//=============================================================================
// ST10_Flow15_FRobot_3.scl
// 1:1 CONVERSION FROM TIA PORTAL V18 GRAPH XML
// Generated: 2026-02-02
//=============================================================================

TYPE
    E_STEP_ST10_Flow15_FRobot_3 : (
        STEP_ST10_Flow15_FRobot_3_WaitRobotGripStatus := 360,
        STEP_ST10_Flow15_FRobot_3_WaitRobotFinish_4 := 356,
        STEP_ST10_Flow15_FRobot_3_ReqRobotToHomePos := 707,
        STEP_ST10_Flow15_FRobot_3_WaitRobotGripStatus_6 := 378,
        STEP_ST10_Flow15_FRobot_3_Tablecode_ScanFinish := 149,
        STEP_ST10_Flow15_FRobot_3_Open_NG_BOX_REQUESTED_ := 111,
        STEP_ST10_Flow15_FRobot_3_RobotReady_ := 311,
        STEP_ST10_Flow15_FRobot_3_PickPalletProcess := 250,
        STEP_ST10_Flow15_FRobot_3_WaitRobotFinish_9 := 371,
        STEP_ST10_Flow15_FRobot_3_WaitRobotReachPos4 := 318,
        STEP_ST10_Flow15_FRobot_3_WaitRobotStartHome := 383,
        STEP_ST10_Flow15_FRobot_3_RobotAutoCycle := 329,
        STEP_ST10_Flow15_FRobot_3_NG3_PutProcessFinish := 849,
        STEP_ST10_Flow15_FRobot_3_WaitRobotFinish_8 := 368,
        STEP_ST10_Flow15_FRobot_3_RobotScanGripperReachPos4 := 341,
        STEP_ST10_Flow15_FRobot_3_Step930 := 930,
        STEP_ST10_Flow15_FRobot_3_DataMove_6 := 266,
        STEP_ST10_Flow15_FRobot_3_ScanRing := 135,
        STEP_ST10_Flow15_FRobot_3_WaitRobotFinish_11 := 377,
        STEP_ST10_Flow15_FRobot_3_WaitRobotGripHaveStatus_2 := 348,
        STEP_ST10_Flow15_FRobot_3_WaitRobotGripStatus_3 := 369,
        STEP_ST10_Flow15_FRobot_3_S9 := 9,
        STEP_ST10_Flow15_FRobot_3_PartOKStatus := 249,
        STEP_ST10_Flow15_FRobot_3_WaitGripperPos3ScanFinish := 340,
        STEP_ST10_Flow15_FRobot_3_WaitBrakeTestFinish := 921,
        STEP_ST10_Flow15_FRobot_3_NG2_PutProcessFinish := 799,
        STEP_ST10_Flow15_FRobot_3_PressPick := 150,
        STEP_ST10_Flow15_FRobot_3_DataMove_2 := 257,
        STEP_ST10_Flow15_FRobot_3_DataMove_5 := 264,
        STEP_ST10_Flow15_FRobot_3_WaitRobotFinish := 327,
        STEP_ST10_Flow15_FRobot_3_StartRobotGluePut := 367,
        STEP_ST10_Flow15_FRobot_3_NG2Put_1Press_Glue := 160,
        STEP_ST10_Flow15_FRobot_3_F15_Initial := 1,
        STEP_ST10_Flow15_FRobot_3_BrakeTestFinish := 929,
        STEP_ST10_Flow15_FRobot_3_StartRobotNG2Put_1 := 373,
        STEP_ST10_Flow15_FRobot_3_NG2Put_2_Magnet := 165,
        STEP_ST10_Flow15_FRobot_3_WaitPos4ScanFinish := 319,
        STEP_ST10_Flow15_FRobot_3_PartOKStatus_1 := 273,
        STEP_ST10_Flow15_FRobot_3_WaitR1HomePosFinsh_1 := 899,
        STEP_ST10_Flow15_FRobot_3_RobotScanGripperReachPos2 := 337,
        STEP_ST10_Flow15_FRobot_3_StartRobotPickGlueNG := 328,
        STEP_ST10_Flow15_FRobot_3_PressRingPutProcessFinish := 599,
        STEP_ST10_Flow15_FRobot_3_StartRobotScanGripperCode := 334,
        STEP_ST10_Flow15_FRobot_3_DataMove_7 := 270,
        STEP_ST10_Flow15_FRobot_3_Maintenance := 131,
        STEP_ST10_Flow15_FRobot_3_Grip1PartStatus := 243,
        STEP_ST10_Flow15_FRobot_3_Grip1SensorError := 381,
        STEP_ST10_Flow15_FRobot_3_WaitMasteringTestFinish := 911,
        STEP_ST10_Flow15_FRobot_3_DataMove_4 := 262,
        STEP_ST10_Flow15_FRobot_3_PressShaftPut := 140,
        STEP_ST10_Flow15_FRobot_3_WaitRobotFinish_5 := 359,
        STEP_ST10_Flow15_FRobot_3_WaitRobotGripHaveStatus := 346,
        STEP_ST10_Flow15_FRobot_3_WaitRobotFinish_1 := 343,
        STEP_ST10_Flow15_FRobot_3_WaitGripperPos1ScanFinish := 336,
        STEP_ST10_Flow15_FRobot_3_RobotStart := 316,
        STEP_ST10_Flow15_FRobot_3_WaitPos2ScanFinish := 312,
        STEP_ST10_Flow15_FRobot_3_WaitRobotReachPos2 := 313,
        STEP_ST10_Flow15_FRobot_3_RobotHome := 317,
        STEP_ST10_Flow15_FRobot_3_WaitGripperPos4ScanFinish := 342,
        STEP_ST10_Flow15_FRobot_3_WaitScanCompletely := 247,
        STEP_ST10_Flow15_FRobot_3_PickGlueNGFinish_1 := 349,
        STEP_ST10_Flow15_FRobot_3_Grip2PartStatus := 244,
        STEP_ST10_Flow15_FRobot_3_WaitRobotFinish_3 := 353,
        STEP_ST10_Flow15_FRobot_3_WaitRobotGripStatus_1 := 363,
        STEP_ST10_Flow15_FRobot_3_NG2Put_3_Ring := 170,
        STEP_ST10_Flow15_FRobot_3_FlagReset := 272,
        STEP_ST10_Flow15_FRobot_3_WaitRobotGripStatus_2 := 366,
        STEP_ST10_Flow15_FRobot_3_WaitRobotFinish_6 := 362,
        STEP_ST10_Flow15_FRobot_3_Gripe2StatusAlarm := 332,
        STEP_ST10_Flow15_FRobot_3_DataMove_8 := 271,
        STEP_ST10_Flow15_FRobot_3_StartRobotPickTable := 352,
        STEP_ST10_Flow15_FRobot_3_ScanStart := 246,
        STEP_ST10_Flow15_FRobot_3_PickGlueNGReq := 120,
        STEP_ST10_Flow15_FRobot_3_RobotSpeed := 4,
        STEP_ST10_Flow15_FRobot_3_StartRobotPressPick := 364,
        STEP_ST10_Flow15_FRobot_3_MES_Online__offline_ := 385,
        STEP_ST10_Flow15_FRobot_3_S10_InitialFinish := 10,
        STEP_ST10_Flow15_FRobot_3_PickMagnScanNGBufferFinish := 399,
        STEP_ST10_Flow15_FRobot_3_RobotScanGripperReachPos3 := 339,
        STEP_ST10_Flow15_FRobot_3_GripStatusCheck := 330,
        STEP_ST10_Flow15_FRobot_3_ScanRingProcess := 450,
        STEP_ST10_Flow15_FRobot_3_S3 := 3,
        STEP_ST10_Flow15_FRobot_3_NG_2_PutProcess := 750,
        STEP_ST10_Flow15_FRobot_3_WaitRobotFinish_10 := 374,
        STEP_ST10_Flow15_FRobot_3_GluePutProcess := 650,
        STEP_ST10_Flow15_FRobot_3_PickTableProcessFinish := 449,
        STEP_ST10_Flow15_FRobot_3_DataClear := 252,
        STEP_ST10_Flow15_FRobot_3_Data_Clear_2 := 258,
        STEP_ST10_Flow15_FRobot_3_PickMagnetNGReqPick := 125,
        STEP_ST10_Flow15_FRobot_3_PressRingPutProcess := 550,
        STEP_ST10_Flow15_FRobot_3_WaitRobotFinish_2 := 345,
        STEP_ST10_Flow15_FRobot_3_PickTableProcess := 400,
        STEP_ST10_Flow15_FRobot_3_WaitRobotGripHaveStatus_3 := 354,
        STEP_ST10_Flow15_FRobot_3_NG_PutProcess := 700,
        STEP_ST10_Flow15_FRobot_3_StartRobotNGPut := 370,
        STEP_ST10_Flow15_FRobot_3_WaitRobotReachPos3 := 314,
        STEP_ST10_Flow15_FRobot_3_Maintenance_Pos := 850,
        STEP_ST10_Flow15_FRobot_3_PressPickProcess := 600,
        STEP_ST10_Flow15_FRobot_3_Data_Clear_9 := 269,
        STEP_ST10_Flow15_FRobot_3_PressPickProcessFinish_ := 649,
        STEP_ST10_Flow15_FRobot_3_WaitGripperPos2ScanFinish := 338,
        STEP_ST10_Flow15_FRobot_3_Tablecode_Scan := 200,
        STEP_ST10_Flow15_FRobot_3_MasteringTest_Req := 910,
        STEP_ST10_Flow15_FRobot_3_ProcessStart := 100,
        STEP_ST10_Flow15_FRobot_3_PartNGStatus := 251,
        STEP_ST10_Flow15_FRobot_3_Data_Clear_8 := 268,
        STEP_ST10_Flow15_FRobot_3_RobotManuallyMoved_ := 384,
        STEP_ST10_Flow15_FRobot_3_S5_MESInitial := 5,
        STEP_ST10_Flow15_FRobot_3_WaitRobotHomeRequest := 706,
        STEP_ST10_Flow15_FRobot_3_Masref_test := 132,
        STEP_ST10_Flow15_FRobot_3_BrakeTest_Req := 920,
        STEP_ST10_Flow15_FRobot_3_WaitRobotGripStatus_5 := 375,
        STEP_ST10_Flow15_FRobot_3_Data_Clear_4 := 261,
        STEP_ST10_Flow15_FRobot_3_ScanRingProcessFinish := 499,
        STEP_ST10_Flow15_FRobot_3_StartRobotPressShaftPut := 358,
        STEP_ST10_Flow15_FRobot_3_WaitPos1ScanFinish := 310,
        STEP_ST10_Flow15_FRobot_3_StartRobotScanFixtureCode := 308,
        STEP_ST10_Flow15_FRobot_3_StartRobotPickMagnScanNG := 344,
        STEP_ST10_Flow15_FRobot_3_ScanFixtureCode := 110,
        STEP_ST10_Flow15_FRobot_3_PressRingPut := 145,
        STEP_ST10_Flow15_FRobot_3_PickPallet := 115,
        STEP_ST10_Flow15_FRobot_3_WaitPos3ScanFinish := 315,
        STEP_ST10_Flow15_FRobot_3_WaitRobotReachScanPos := 357,
        STEP_ST10_Flow15_FRobot_3_StartRobotPressRingPut := 361,
        STEP_ST10_Flow15_FRobot_3_ReqRobotToMantenPos_1 := 704,
        STEP_ST10_Flow15_FRobot_3_PickTable := 130,
        STEP_ST10_Flow15_FRobot_3_DataMove_3 := 260,
        STEP_ST10_Flow15_FRobot_3_PickGlueNGProcess := 300,
        STEP_ST10_Flow15_FRobot_3_StartRobotPickPalletShaft := 326,
        STEP_ST10_Flow15_FRobot_3_NG1_PutProcessFinish := 749,
        STEP_ST10_Flow15_FRobot_3_OKPut := 155,
        STEP_ST10_Flow15_FRobot_3_PickPalletFinish := 299,
        STEP_ST10_Flow15_FRobot_3_MagnScanNGProcess := 350,
        STEP_ST10_Flow15_FRobot_3_OKPutProcessFinish := 699,
        STEP_ST10_Flow15_FRobot_3_StartRobotScanRing := 355,
        STEP_ST10_Flow15_FRobot_3_PressShaftPutProcessFinish := 549,
        STEP_ST10_Flow15_FRobot_3_DataMove_1 := 255,
        STEP_ST10_Flow15_FRobot_3_Grip2SensorError := 382,
        STEP_ST10_Flow15_FRobot_3_DataMove := 253,
        STEP_ST10_Flow15_FRobot_3_MasteringTestFinish := 919,
        STEP_ST10_Flow15_FRobot_3_S_900 := 900,
        STEP_ST10_Flow15_FRobot_3_WaitRobotReachPos1 := 309,
        STEP_ST10_Flow15_FRobot_3_RobotScanGripperReachPos1 := 335,
        STEP_ST10_Flow15_FRobot_3_Data_Clear_7 := 267,
        STEP_ST10_Flow15_FRobot_3_WaitR1MaintenPosFinsh_1 := 705,
        STEP_ST10_Flow15_FRobot_3_PressShaftPutProcess := 500,
        STEP_ST10_Flow15_FRobot_3_StartRobotNG3Put := 376,
        STEP_ST10_Flow15_FRobot_3_RobotTaskSelect := 333,
        STEP_ST10_Flow15_FRobot_3_NG_3_PutProcess := 800,
        STEP_ST10_Flow15_FRobot_3_Brake_Test := 133,
        STEP_ST10_Flow15_FRobot_3_WaitRobotFinish_7 := 365,
        STEP_ST10_Flow15_FRobot_3_Gripe1StatusAlarm := 331,
        STEP_ST10_Flow15_FRobot_3_WaitRobotGripStatus_4 := 372,
        STEP_ST10_Flow15_FRobot_3_Data_Clear_6 := 265,
        STEP_ST10_Flow15_FRobot_3_S2 := 2,
        STEP_ST10_Flow15_FRobot_3_CheckScanReady := 245,
        STEP_ST10_Flow15_FRobot_3_S8 := 8,
        STEP_ST10_Flow15_FRobot_3_CodeMove := 248,
        STEP_ST10_Flow15_FRobot_3_WaitRobotGripHaveStatus_1 := 347,
    ) INT := 1;
END_TYPE

CONST
    STEP_ST10_Flow15_FRobot_3_WaitRobotGripStatus := 360;
    STEP_ST10_Flow15_FRobot_3_WaitRobotFinish_4 := 356;
    STEP_ST10_Flow15_FRobot_3_ReqRobotToHomePos := 707;
    STEP_ST10_Flow15_FRobot_3_WaitRobotGripStatus_6 := 378;
    STEP_ST10_Flow15_FRobot_3_Tablecode_ScanFinish := 149;
    STEP_ST10_Flow15_FRobot_3_Open_NG_BOX_REQUESTED_ := 111;
    STEP_ST10_Flow15_FRobot_3_RobotReady_ := 311;
    STEP_ST10_Flow15_FRobot_3_PickPalletProcess := 250;
    STEP_ST10_Flow15_FRobot_3_WaitRobotFinish_9 := 371;
    STEP_ST10_Flow15_FRobot_3_WaitRobotReachPos4 := 318;
    STEP_ST10_Flow15_FRobot_3_WaitRobotStartHome := 383;
    STEP_ST10_Flow15_FRobot_3_RobotAutoCycle := 329;
    STEP_ST10_Flow15_FRobot_3_NG3_PutProcessFinish := 849;
    STEP_ST10_Flow15_FRobot_3_WaitRobotFinish_8 := 368;
    STEP_ST10_Flow15_FRobot_3_RobotScanGripperReachPos4 := 341;
    STEP_ST10_Flow15_FRobot_3_Step930 := 930;
    STEP_ST10_Flow15_FRobot_3_DataMove_6 := 266;
    STEP_ST10_Flow15_FRobot_3_ScanRing := 135;
    STEP_ST10_Flow15_FRobot_3_WaitRobotFinish_11 := 377;
    STEP_ST10_Flow15_FRobot_3_WaitRobotGripHaveStatus_2 := 348;
    STEP_ST10_Flow15_FRobot_3_WaitRobotGripStatus_3 := 369;
    STEP_ST10_Flow15_FRobot_3_S9 := 9;
    STEP_ST10_Flow15_FRobot_3_PartOKStatus := 249;
    STEP_ST10_Flow15_FRobot_3_WaitGripperPos3ScanFinish := 340;
    STEP_ST10_Flow15_FRobot_3_WaitBrakeTestFinish := 921;
    STEP_ST10_Flow15_FRobot_3_NG2_PutProcessFinish := 799;
    STEP_ST10_Flow15_FRobot_3_PressPick := 150;
    STEP_ST10_Flow15_FRobot_3_DataMove_2 := 257;
    STEP_ST10_Flow15_FRobot_3_DataMove_5 := 264;
    STEP_ST10_Flow15_FRobot_3_WaitRobotFinish := 327;
    STEP_ST10_Flow15_FRobot_3_StartRobotGluePut := 367;
    STEP_ST10_Flow15_FRobot_3_NG2Put_1Press_Glue := 160;
    STEP_ST10_Flow15_FRobot_3_F15_Initial := 1;
    STEP_ST10_Flow15_FRobot_3_BrakeTestFinish := 929;
    STEP_ST10_Flow15_FRobot_3_StartRobotNG2Put_1 := 373;
    STEP_ST10_Flow15_FRobot_3_NG2Put_2_Magnet := 165;
    STEP_ST10_Flow15_FRobot_3_WaitPos4ScanFinish := 319;
    STEP_ST10_Flow15_FRobot_3_PartOKStatus_1 := 273;
    STEP_ST10_Flow15_FRobot_3_WaitR1HomePosFinsh_1 := 899;
    STEP_ST10_Flow15_FRobot_3_RobotScanGripperReachPos2 := 337;
    STEP_ST10_Flow15_FRobot_3_StartRobotPickGlueNG := 328;
    STEP_ST10_Flow15_FRobot_3_PressRingPutProcessFinish := 599;
    STEP_ST10_Flow15_FRobot_3_StartRobotScanGripperCode := 334;
    STEP_ST10_Flow15_FRobot_3_DataMove_7 := 270;
    STEP_ST10_Flow15_FRobot_3_Maintenance := 131;
    STEP_ST10_Flow15_FRobot_3_Grip1PartStatus := 243;
    STEP_ST10_Flow15_FRobot_3_Grip1SensorError := 381;
    STEP_ST10_Flow15_FRobot_3_WaitMasteringTestFinish := 911;
    STEP_ST10_Flow15_FRobot_3_DataMove_4 := 262;
    STEP_ST10_Flow15_FRobot_3_PressShaftPut := 140;
    STEP_ST10_Flow15_FRobot_3_WaitRobotFinish_5 := 359;
    STEP_ST10_Flow15_FRobot_3_WaitRobotGripHaveStatus := 346;
    STEP_ST10_Flow15_FRobot_3_WaitRobotFinish_1 := 343;
    STEP_ST10_Flow15_FRobot_3_WaitGripperPos1ScanFinish := 336;
    STEP_ST10_Flow15_FRobot_3_RobotStart := 316;
    STEP_ST10_Flow15_FRobot_3_WaitPos2ScanFinish := 312;
    STEP_ST10_Flow15_FRobot_3_WaitRobotReachPos2 := 313;
    STEP_ST10_Flow15_FRobot_3_RobotHome := 317;
    STEP_ST10_Flow15_FRobot_3_WaitGripperPos4ScanFinish := 342;
    STEP_ST10_Flow15_FRobot_3_WaitScanCompletely := 247;
    STEP_ST10_Flow15_FRobot_3_PickGlueNGFinish_1 := 349;
    STEP_ST10_Flow15_FRobot_3_Grip2PartStatus := 244;
    STEP_ST10_Flow15_FRobot_3_WaitRobotFinish_3 := 353;
    STEP_ST10_Flow15_FRobot_3_WaitRobotGripStatus_1 := 363;
    STEP_ST10_Flow15_FRobot_3_NG2Put_3_Ring := 170;
    STEP_ST10_Flow15_FRobot_3_FlagReset := 272;
    STEP_ST10_Flow15_FRobot_3_WaitRobotGripStatus_2 := 366;
    STEP_ST10_Flow15_FRobot_3_WaitRobotFinish_6 := 362;
    STEP_ST10_Flow15_FRobot_3_Gripe2StatusAlarm := 332;
    STEP_ST10_Flow15_FRobot_3_DataMove_8 := 271;
    STEP_ST10_Flow15_FRobot_3_StartRobotPickTable := 352;
    STEP_ST10_Flow15_FRobot_3_ScanStart := 246;
    STEP_ST10_Flow15_FRobot_3_PickGlueNGReq := 120;
    STEP_ST10_Flow15_FRobot_3_RobotSpeed := 4;
    STEP_ST10_Flow15_FRobot_3_StartRobotPressPick := 364;
    STEP_ST10_Flow15_FRobot_3_MES_Online__offline_ := 385;
    STEP_ST10_Flow15_FRobot_3_S10_InitialFinish := 10;
    STEP_ST10_Flow15_FRobot_3_PickMagnScanNGBufferFinish := 399;
    STEP_ST10_Flow15_FRobot_3_RobotScanGripperReachPos3 := 339;
    STEP_ST10_Flow15_FRobot_3_GripStatusCheck := 330;
    STEP_ST10_Flow15_FRobot_3_ScanRingProcess := 450;
    STEP_ST10_Flow15_FRobot_3_S3 := 3;
    STEP_ST10_Flow15_FRobot_3_NG_2_PutProcess := 750;
    STEP_ST10_Flow15_FRobot_3_WaitRobotFinish_10 := 374;
    STEP_ST10_Flow15_FRobot_3_GluePutProcess := 650;
    STEP_ST10_Flow15_FRobot_3_PickTableProcessFinish := 449;
    STEP_ST10_Flow15_FRobot_3_DataClear := 252;
    STEP_ST10_Flow15_FRobot_3_Data_Clear_2 := 258;
    STEP_ST10_Flow15_FRobot_3_PickMagnetNGReqPick := 125;
    STEP_ST10_Flow15_FRobot_3_PressRingPutProcess := 550;
    STEP_ST10_Flow15_FRobot_3_WaitRobotFinish_2 := 345;
    STEP_ST10_Flow15_FRobot_3_PickTableProcess := 400;
    STEP_ST10_Flow15_FRobot_3_WaitRobotGripHaveStatus_3 := 354;
    STEP_ST10_Flow15_FRobot_3_NG_PutProcess := 700;
    STEP_ST10_Flow15_FRobot_3_StartRobotNGPut := 370;
    STEP_ST10_Flow15_FRobot_3_WaitRobotReachPos3 := 314;
    STEP_ST10_Flow15_FRobot_3_Maintenance_Pos := 850;
    STEP_ST10_Flow15_FRobot_3_PressPickProcess := 600;
    STEP_ST10_Flow15_FRobot_3_Data_Clear_9 := 269;
    STEP_ST10_Flow15_FRobot_3_PressPickProcessFinish_ := 649;
    STEP_ST10_Flow15_FRobot_3_WaitGripperPos2ScanFinish := 338;
    STEP_ST10_Flow15_FRobot_3_Tablecode_Scan := 200;
    STEP_ST10_Flow15_FRobot_3_MasteringTest_Req := 910;
    STEP_ST10_Flow15_FRobot_3_ProcessStart := 100;
    STEP_ST10_Flow15_FRobot_3_PartNGStatus := 251;
    STEP_ST10_Flow15_FRobot_3_Data_Clear_8 := 268;
    STEP_ST10_Flow15_FRobot_3_RobotManuallyMoved_ := 384;
    STEP_ST10_Flow15_FRobot_3_S5_MESInitial := 5;
    STEP_ST10_Flow15_FRobot_3_WaitRobotHomeRequest := 706;
    STEP_ST10_Flow15_FRobot_3_Masref_test := 132;
    STEP_ST10_Flow15_FRobot_3_BrakeTest_Req := 920;
    STEP_ST10_Flow15_FRobot_3_WaitRobotGripStatus_5 := 375;
    STEP_ST10_Flow15_FRobot_3_Data_Clear_4 := 261;
    STEP_ST10_Flow15_FRobot_3_ScanRingProcessFinish := 499;
    STEP_ST10_Flow15_FRobot_3_StartRobotPressShaftPut := 358;
    STEP_ST10_Flow15_FRobot_3_WaitPos1ScanFinish := 310;
    STEP_ST10_Flow15_FRobot_3_StartRobotScanFixtureCode := 308;
    STEP_ST10_Flow15_FRobot_3_StartRobotPickMagnScanNG := 344;
    STEP_ST10_Flow15_FRobot_3_ScanFixtureCode := 110;
    STEP_ST10_Flow15_FRobot_3_PressRingPut := 145;
    STEP_ST10_Flow15_FRobot_3_PickPallet := 115;
    STEP_ST10_Flow15_FRobot_3_WaitPos3ScanFinish := 315;
    STEP_ST10_Flow15_FRobot_3_WaitRobotReachScanPos := 357;
    STEP_ST10_Flow15_FRobot_3_StartRobotPressRingPut := 361;
    STEP_ST10_Flow15_FRobot_3_ReqRobotToMantenPos_1 := 704;
    STEP_ST10_Flow15_FRobot_3_PickTable := 130;
    STEP_ST10_Flow15_FRobot_3_DataMove_3 := 260;
    STEP_ST10_Flow15_FRobot_3_PickGlueNGProcess := 300;
    STEP_ST10_Flow15_FRobot_3_StartRobotPickPalletShaft := 326;
    STEP_ST10_Flow15_FRobot_3_NG1_PutProcessFinish := 749;
    STEP_ST10_Flow15_FRobot_3_OKPut := 155;
    STEP_ST10_Flow15_FRobot_3_PickPalletFinish := 299;
    STEP_ST10_Flow15_FRobot_3_MagnScanNGProcess := 350;
    STEP_ST10_Flow15_FRobot_3_OKPutProcessFinish := 699;
    STEP_ST10_Flow15_FRobot_3_StartRobotScanRing := 355;
    STEP_ST10_Flow15_FRobot_3_PressShaftPutProcessFinish := 549;
    STEP_ST10_Flow15_FRobot_3_DataMove_1 := 255;
    STEP_ST10_Flow15_FRobot_3_Grip2SensorError := 382;
    STEP_ST10_Flow15_FRobot_3_DataMove := 253;
    STEP_ST10_Flow15_FRobot_3_MasteringTestFinish := 919;
    STEP_ST10_Flow15_FRobot_3_S_900 := 900;
    STEP_ST10_Flow15_FRobot_3_WaitRobotReachPos1 := 309;
    STEP_ST10_Flow15_FRobot_3_RobotScanGripperReachPos1 := 335;
    STEP_ST10_Flow15_FRobot_3_Data_Clear_7 := 267;
    STEP_ST10_Flow15_FRobot_3_WaitR1MaintenPosFinsh_1 := 705;
    STEP_ST10_Flow15_FRobot_3_PressShaftPutProcess := 500;
    STEP_ST10_Flow15_FRobot_3_StartRobotNG3Put := 376;
    STEP_ST10_Flow15_FRobot_3_RobotTaskSelect := 333;
    STEP_ST10_Flow15_FRobot_3_NG_3_PutProcess := 800;
    STEP_ST10_Flow15_FRobot_3_Brake_Test := 133;
    STEP_ST10_Flow15_FRobot_3_WaitRobotFinish_7 := 365;
    STEP_ST10_Flow15_FRobot_3_Gripe1StatusAlarm := 331;
    STEP_ST10_Flow15_FRobot_3_WaitRobotGripStatus_4 := 372;
    STEP_ST10_Flow15_FRobot_3_Data_Clear_6 := 265;
    STEP_ST10_Flow15_FRobot_3_S2 := 2;
    STEP_ST10_Flow15_FRobot_3_CheckScanReady := 245;
    STEP_ST10_Flow15_FRobot_3_S8 := 8;
    STEP_ST10_Flow15_FRobot_3_CodeMove := 248;
    STEP_ST10_Flow15_FRobot_3_WaitRobotGripHaveStatus_1 := 347;
END_CONST

FUNCTION_BLOCK "ST10_Flow15_FRobot_3_1to1"
{ S7_Optimized_Access := 'TRUE' }
VERSION : 1.0

VAR_INPUT
    iSysInface : "RCS_SysComInterface_V1";
END_VAR

VAR_IN_OUT
    ioPM_Inface : "RCS_PMInterface_V1";
    ioStatus : Int;
END_VAR

VAR_OUTPUT
    oAlarmID : Int;
END_VAR

VAR
    State : INT := 1;
    act_InitialRun : Bool;
    act_InitialOK : Bool;
    act_WaitRunning : Bool;
    act_Running : Bool;
    act_ProcessComplete : Bool;
    act_ProcessStart : Bool;
    act_UnPause : Bool;
    bError : Bool;
    wErrorID : Word;
END_VAR

BEGIN
    //======================================================================
    // STATE MACHINE - Inline Transition Conditions
    //======================================================================

    CASE #State OF

        // ===========================================
        // STEP 360: WaitRobotGripStatus
        // ===========================================
        STEP_ST10_Flow15_FRobot_3_WaitRobotGripStatus:
            // No actions in XML

            // Transition to next step: 356
            IF TRUE THEN  // Sequential transition - review XML for actual condition
                #State := STEP_ST10_Flow15_FRobot_3_WaitRobotFinish_4;
            END_IF;

        // ===========================================
        // STEP 356: WaitRobotFinish_4
        // ===========================================
        STEP_ST10_Flow15_FRobot_3_WaitRobotFinish_4:
            // Action Qualifier=N
            // Token: "KukaRobot3_CtrlDB".sPLCtoROB.User.Cycle.DI262_ScanRingComplete
            "KukaRobot3_CtrlDB".sPLCtoROB.User.Cycle.DI262_ScanRingComplete;

            // Transition to next step: 707
            IF TRUE THEN  // Sequential transition - review XML for actual condition
                #State := STEP_ST10_Flow15_FRobot_3_ReqRobotToHomePos;
            END_IF;

        // ===========================================
        // STEP 707: ReqRobotToHomePos
        // ===========================================
        STEP_ST10_Flow15_FRobot_3_ReqRobotToHomePos:
            // Action Qualifier=N
            // Token: "KukaRobot3_CtrlDB".sPLCtoROB.User.Cycle.DI300_HomeRequest
            "KukaRobot3_CtrlDB".sPLCtoROB.User.Cycle.DI300_HomeRequest;

            // Transition to next step: 378
            IF TRUE THEN  // Sequential transition - review XML for actual condition
                #State := STEP_ST10_Flow15_FRobot_3_WaitRobotGripStatus_6;
            END_IF;

        // ===========================================
        // STEP 378: WaitRobotGripStatus_6
        // ===========================================
        STEP_ST10_Flow15_FRobot_3_WaitRobotGripStatus_6:
            // No actions in XML

            // Transition to next step: 149
            IF TRUE THEN  // Sequential transition - review XML for actual condition
                #State := STEP_ST10_Flow15_FRobot_3_Tablecode_ScanFinish;
            END_IF;

        // ===========================================
        // STEP 149: Tablecode ScanFinish
        // ===========================================
        STEP_ST10_Flow15_FRobot_3_Tablecode_ScanFinish:
            // Action Qualifier=S
            // Token: #ioPM_Inface.ProcessComplete
            #ioPM_Inface.ProcessComplete := TRUE;
            // Action Qualifier=R
            // Token: #ioPM_Inface.ProcessStart
            #ioPM_Inface.ProcessStart := FALSE;

            // Transition to next step: 111
            IF TRUE THEN  // Sequential transition - review XML for actual condition
                #State := STEP_ST10_Flow15_FRobot_3_Open_NG_BOX_REQUESTED_;
            END_IF;

        // ===========================================
        // STEP 111: Open NG BOX REQUESTED?
        // ===========================================
        STEP_ST10_Flow15_FRobot_3_Open_NG_BOX_REQUESTED_:
            // No actions in XML

            // Transition to next step: 311
            IF TRUE THEN  // Sequential transition - review XML for actual condition
                #State := STEP_ST10_Flow15_FRobot_3_RobotReady_;
            END_IF;

        // ===========================================
        // STEP 311: RobotReady?
        // ===========================================
        STEP_ST10_Flow15_FRobot_3_RobotReady_:
            // No actions in XML

            // Transition to next step: 250
            IF TRUE THEN  // Sequential transition - review XML for actual condition
                #State := STEP_ST10_Flow15_FRobot_3_PickPalletProcess;
            END_IF;

        // ===========================================
        // STEP 250: PickPalletProcess
        // ===========================================
        STEP_ST10_Flow15_FRobot_3_PickPalletProcess:
            // No actions in XML

            // Transition to next step: 371
            IF TRUE THEN  // Sequential transition - review XML for actual condition
                #State := STEP_ST10_Flow15_FRobot_3_WaitRobotFinish_9;
            END_IF;

        // ===========================================
        // STEP 371: WaitRobotFinish_9
        // ===========================================
        STEP_ST10_Flow15_FRobot_3_WaitRobotFinish_9:
            // No actions in XML

            // Transition to next step: 318
            IF TRUE THEN  // Sequential transition - review XML for actual condition
                #State := STEP_ST10_Flow15_FRobot_3_WaitRobotReachPos4;
            END_IF;

        // ===========================================
        // STEP 318: WaitRobotReachPos4
        // ===========================================
        STEP_ST10_Flow15_FRobot_3_WaitRobotReachPos4:
            // No actions in XML

            // Transition to next step: 383
            IF TRUE THEN  // Sequential transition - review XML for actual condition
                #State := STEP_ST10_Flow15_FRobot_3_WaitRobotStartHome;
            END_IF;

        // ===========================================
        // STEP 383: WaitRobotStartHome
        // ===========================================
        STEP_ST10_Flow15_FRobot_3_WaitRobotStartHome:
            // No actions in XML

            // Transition to next step: 329
            IF TRUE THEN  // Sequential transition - review XML for actual condition
                #State := STEP_ST10_Flow15_FRobot_3_RobotAutoCycle;
            END_IF;

        // ===========================================
        // STEP 329: RobotAutoCycle
        // ===========================================
        STEP_ST10_Flow15_FRobot_3_RobotAutoCycle:
            // Action Qualifier=N
            // Token: "KukaRobot3_CtrlDB".ioStartAutoCycle
            "KukaRobot3_CtrlDB".ioStartAutoCycle;

            // Transition to next step: 849
            IF TRUE THEN  // Sequential transition - review XML for actual condition
                #State := STEP_ST10_Flow15_FRobot_3_NG3_PutProcessFinish;
            END_IF;

        // ===========================================
        // STEP 849: NG3 PutProcessFinish
        // ===========================================
        STEP_ST10_Flow15_FRobot_3_NG3_PutProcessFinish:
            // Action Qualifier=S
            // Token: #ioPM_Inface.ProcessComplete
            #ioPM_Inface.ProcessComplete := TRUE;
            // Action Qualifier=R
            // Token: #ioPM_Inface.ProcessStart
            #ioPM_Inface.ProcessStart := FALSE;

            // Transition to next step: 368
            IF TRUE THEN  // Sequential transition - review XML for actual condition
                #State := STEP_ST10_Flow15_FRobot_3_WaitRobotFinish_8;
            END_IF;

        // ===========================================
        // STEP 368: WaitRobotFinish_8
        // ===========================================
        STEP_ST10_Flow15_FRobot_3_WaitRobotFinish_8:
            // No actions in XML

            // Transition to next step: 341
            IF TRUE THEN  // Sequential transition - review XML for actual condition
                #State := STEP_ST10_Flow15_FRobot_3_RobotScanGripperReachPos4;
            END_IF;

        // ===========================================
        // STEP 341: RobotScanGripperReachPos4
        // ===========================================
        STEP_ST10_Flow15_FRobot_3_RobotScanGripperReachPos4:
            // No actions in XML

            // Transition to next step: 930
            IF TRUE THEN  // Sequential transition - review XML for actual condition
                #State := STEP_ST10_Flow15_FRobot_3_Step930;
            END_IF;

        // ===========================================
        // STEP 930: Step930
        // ===========================================
        STEP_ST10_Flow15_FRobot_3_Step930:
            // Action Qualifier=N
            // Token: //"AutoProcessData".F_Robot3Grip1.PartStatus:=444
            //"AutoProcessData".F_Robot3Grip1.PartStatus:=444;

            // Transition to next step: 266
            IF TRUE THEN  // Sequential transition - review XML for actual condition
                #State := STEP_ST10_Flow15_FRobot_3_DataMove_6;
            END_IF;

        // ===========================================
        // STEP 266: DataMove_6
        // ===========================================
        STEP_ST10_Flow15_FRobot_3_DataMove_6:
            // Action Qualifier=N
            // Token: //"AutoProcessData_Buffer".DataBuffer["AutoProcessData".GlobalData.DataIndex]:="AutoProcessData".F_Robot3Grip1
            //"AutoProcessData_Buffer".DataBuffer["AutoProcessData".GlobalData.DataIndex]:="AutoProcessData".F_Robot3Grip1;
            // Action Qualifier=N
            // Token: //"AutoProcessData".GlobalData.DataIndex:="AutoProcessData".GlobalData.DataIndex+1
            //"AutoProcessData".GlobalData.DataIndex:="AutoProcessData".GlobalData.DataIndex+1;

            // Transition to next step: 135
            IF TRUE THEN  // Sequential transition - review XML for actual condition
                #State := STEP_ST10_Flow15_FRobot_3_ScanRing;
            END_IF;

        // ===========================================
        // STEP 135: ScanRing
        // ===========================================
        STEP_ST10_Flow15_FRobot_3_ScanRing:
            // Action Qualifier=R
            // Token: #ioPM_Inface.ProcessComplete
            #ioPM_Inface.ProcessComplete := FALSE;
            // Action Qualifier=S
            // Token: #ioPM_Inface.ProcessStart
            #ioPM_Inface.ProcessStart := TRUE;

            // Transition to next step: 377
            IF TRUE THEN  // Sequential transition - review XML for actual condition
                #State := STEP_ST10_Flow15_FRobot_3_WaitRobotFinish_11;
            END_IF;

        // ===========================================
        // STEP 377: WaitRobotFinish_11
        // ===========================================
        STEP_ST10_Flow15_FRobot_3_WaitRobotFinish_11:
            // No actions in XML

            // Transition to next step: 348
            IF TRUE THEN  // Sequential transition - review XML for actual condition
                #State := STEP_ST10_Flow15_FRobot_3_WaitRobotGripHaveStatus_2;
            END_IF;

        // ===========================================
        // STEP 348: WaitRobotGripHaveStatus_2
        // ===========================================
        STEP_ST10_Flow15_FRobot_3_WaitRobotGripHaveStatus_2:
            // No actions in XML

            // Transition to next step: 369
            IF TRUE THEN  // Sequential transition - review XML for actual condition
                #State := STEP_ST10_Flow15_FRobot_3_WaitRobotGripStatus_3;
            END_IF;

        // ===========================================
        // STEP 369: WaitRobotGripStatus_3
        // ===========================================
        STEP_ST10_Flow15_FRobot_3_WaitRobotGripStatus_3:
            // No actions in XML

            // Transition to next step: 9
            IF TRUE THEN  // Sequential transition - review XML for actual condition
                #State := STEP_ST10_Flow15_FRobot_3_S9;
            END_IF;

        // ===========================================
        // STEP 9: S9
        // ===========================================
        STEP_ST10_Flow15_FRobot_3_S9:
            // No actions in XML

            // Transition to next step: 249
            IF TRUE THEN  // Sequential transition - review XML for actual condition
                #State := STEP_ST10_Flow15_FRobot_3_PartOKStatus;
            END_IF;

        // ===========================================
        // STEP 249: PartOKStatus
        // ===========================================
        STEP_ST10_Flow15_FRobot_3_PartOKStatus:
            // Action Qualifier=N
            // Token: "AutoProcessData".F_Robot3Grip2.PartStatus := 199
            "AutoProcessData".F_Robot3Grip2.PartStatus := 199;

            // Transition to next step: 340
            IF TRUE THEN  // Sequential transition - review XML for actual condition
                #State := STEP_ST10_Flow15_FRobot_3_WaitGripperPos3ScanFinish;
            END_IF;

        // ===========================================
        // STEP 340: WaitGripperPos3ScanFinish
        // ===========================================
        STEP_ST10_Flow15_FRobot_3_WaitGripperPos3ScanFinish:
            // No actions in XML

            // Transition to next step: 921
            IF TRUE THEN  // Sequential transition - review XML for actual condition
                #State := STEP_ST10_Flow15_FRobot_3_WaitBrakeTestFinish;
            END_IF;

        // ===========================================
        // STEP 921: WaitBrakeTestFinish
        // ===========================================
        STEP_ST10_Flow15_FRobot_3_WaitBrakeTestFinish:
            // No actions in XML

            // Transition to next step: 799
            IF TRUE THEN  // Sequential transition - review XML for actual condition
                #State := STEP_ST10_Flow15_FRobot_3_NG2_PutProcessFinish;
            END_IF;

        // ===========================================
        // STEP 799: NG2 PutProcessFinish
        // ===========================================
        STEP_ST10_Flow15_FRobot_3_NG2_PutProcessFinish:
            // Action Qualifier=S
            // Token: #ioPM_Inface.ProcessComplete
            #ioPM_Inface.ProcessComplete := TRUE;
            // Action Qualifier=R
            // Token: #ioPM_Inface.ProcessStart
            #ioPM_Inface.ProcessStart := FALSE;
            // Action Qualifier=N
            // Token: "AutoProcessData".F_Robot3Grip1.PartStatus := 0
            "AutoProcessData".F_Robot3Grip1.PartStatus := 0;

            // Transition to next step: 150
            IF TRUE THEN  // Sequential transition - review XML for actual condition
                #State := STEP_ST10_Flow15_FRobot_3_PressPick;
            END_IF;

        // ===========================================
        // STEP 150: PressPick
        // ===========================================
        STEP_ST10_Flow15_FRobot_3_PressPick:
            // Action Qualifier=R
            // Token: #ioPM_Inface.ProcessComplete
            #ioPM_Inface.ProcessComplete := FALSE;
            // Action Qualifier=S
            // Token: #ioPM_Inface.ProcessStart
            #ioPM_Inface.ProcessStart := TRUE;

            // Transition to next step: 257
            IF TRUE THEN  // Sequential transition - review XML for actual condition
                #State := STEP_ST10_Flow15_FRobot_3_DataMove_2;
            END_IF;

        // ===========================================
        // STEP 257: DataMove_2
        // ===========================================
        STEP_ST10_Flow15_FRobot_3_DataMove_2:
            // Action Qualifier=N, Event="S1"
            // Token: "AutoProcessData".B_Press2 := "AutoProcessData".F_Robot3Grip1
            "AutoProcessData".B_Press2 := "AutoProcessData".F_Robot3Grip1;
            // Action Qualifier=N, Event="S1"
            // Token: "AutoProcessData".F_Robot3Grip1 := "AutoProcessData".ClearData
            "AutoProcessData".F_Robot3Grip1 := "AutoProcessData".ClearData;

            // Transition to next step: 264
            IF TRUE THEN  // Sequential transition - review XML for actual condition
                #State := STEP_ST10_Flow15_FRobot_3_DataMove_5;
            END_IF;

        // ===========================================
        // STEP 264: DataMove_5
        // ===========================================
        STEP_ST10_Flow15_FRobot_3_DataMove_5:
            // Action Qualifier=N, Event="S1"
            // Token: "AutoProcessData_Buffer".DataBuffer["AutoProcessData".GlobalData.DataIndex] := "AutoProcessData".F_Robot3Grip1
            "AutoProcessData_Buffer".DataBuffer["AutoProcessData".GlobalData.DataIndex] := "AutoProcessData".F_Robot3Grip1;
            // Action Qualifier=N, Event="S1"
            // Token: "AutoProcessData".F_Robot3Grip1 := "AutoProcessData".ClearData
            "AutoProcessData".F_Robot3Grip1 := "AutoProcessData".ClearData;
            // Action Qualifier=N, Event="S0"
            // Token: "AutoProcessData".GlobalData.DataIndex := "AutoProcessData".GlobalData.DataIndex + 1
            "AutoProcessData".GlobalData.DataIndex := "AutoProcessData".GlobalData.DataIndex + 1;

            // Transition to next step: 327
            IF TRUE THEN  // Sequential transition - review XML for actual condition
                #State := STEP_ST10_Flow15_FRobot_3_WaitRobotFinish;
            END_IF;

        // ===========================================
        // STEP 327: WaitRobotFinish
        // ===========================================
        STEP_ST10_Flow15_FRobot_3_WaitRobotFinish:
            // No actions in XML

            // Transition to next step: 367
            IF TRUE THEN  // Sequential transition - review XML for actual condition
                #State := STEP_ST10_Flow15_FRobot_3_StartRobotGluePut;
            END_IF;

        // ===========================================
        // STEP 367: StartRobotGluePut
        // ===========================================
        STEP_ST10_Flow15_FRobot_3_StartRobotGluePut:
            // Action Qualifier=N
            // Token: "KukaRobot3_CtrlDB".sPLCtoROB.User.Cycle.DI289_PutOkPartReq
            "KukaRobot3_CtrlDB".sPLCtoROB.User.Cycle.DI289_PutOkPartReq;

            // Transition to next step: 160
            IF TRUE THEN  // Sequential transition - review XML for actual condition
                #State := STEP_ST10_Flow15_FRobot_3_NG2Put_1Press_Glue;
            END_IF;

        // ===========================================
        // STEP 160: NG2Put_1Press/Glue
        // ===========================================
        STEP_ST10_Flow15_FRobot_3_NG2Put_1Press_Glue:
            // Action Qualifier=R
            // Token: #ioPM_Inface.ProcessComplete
            #ioPM_Inface.ProcessComplete := FALSE;
            // Action Qualifier=S
            // Token: #ioPM_Inface.ProcessStart
            #ioPM_Inface.ProcessStart := TRUE;

            // Transition to next step: 1
            IF TRUE THEN  // Sequential transition - review XML for actual condition
                #State := STEP_ST10_Flow15_FRobot_3_F15_Initial;
            END_IF;

        // ===========================================
        // STEP 1: F15_Initial
        // ===========================================
        STEP_ST10_Flow15_FRobot_3_F15_Initial:
            // Action Qualifier=S
            // Token: #ioPM_Inface.InitialRun
            #ioPM_Inface.InitialRun := TRUE;
            // Action Qualifier=R
            // Token: #ioPM_Inface.InitialOK
            #ioPM_Inface.InitialOK := FALSE;
            // Action Qualifier=R
            // Token: #ioPM_Inface.WaitRunning
            #ioPM_Inface.WaitRunning := FALSE;
            // Action Qualifier=R
            // Token: #ioPM_Inface.Running
            #ioPM_Inface.Running := FALSE;
            // Action Qualifier=R
            // Token: #ioPM_Inface.ProcessComplete
            #ioPM_Inface.ProcessComplete := FALSE;
            // Action Qualifier=R
            // Token: #ioPM_Inface.UnPause
            #ioPM_Inface.UnPause := FALSE;
            // Action Qualifier=R
            // Token: "Station_Sys".Cmd.Calibration
            "Station_Sys".Cmd.Calibration := FALSE;
            // Action Qualifier=R
            // Token: "Station_Sys".Cmd.ChangeOver
            "Station_Sys".Cmd.ChangeOver := FALSE;
            // Action Qualifier=N
            // Token: //"ST350_Sys".Cmd.DryRun
            //"ST350_Sys".Cmd.DryRun;
            // Action Qualifier=R
            // Token: "Station_Sys".Cmd.Reserve
            "Station_Sys".Cmd.Reserve := FALSE;
            // Action Qualifier=R
            // Token: "Station_Sys".Cmd.OneCycle
            "Station_Sys".Cmd.OneCycle := FALSE;
            // Action Qualifier=R
            // Token: "AutoProcessControl".Robot_3.Press2PutFlag
            "AutoProcessControl".Robot_3.Press2PutFlag := FALSE;
            // Action Qualifier=R
            // Token: "AutoProcessControl".Robot_3.Press2PickFlag
            "AutoProcessControl".Robot_3.Press2PickFlag := FALSE;
            // Action Qualifier=R
            // Token: "AutoProcessControl".Robot_3.GlueNGPickFlag
            "AutoProcessControl".Robot_3.GlueNGPickFlag := FALSE;
            // Action Qualifier=R
            // Token: "AutoProcessControl".Robot_3.ScanNGPickFlag
            "AutoProcessControl".Robot_3.ScanNGPickFlag := FALSE;
            // Action Qualifier=R
            // Token: "AutoProcessControl".Robot_3.NGPutFlag
            "AutoProcessControl".Robot_3.NGPutFlag := FALSE;
            // Action Qualifier=R
            // Token: #ioPM_Inface.ProcessStart
            #ioPM_Inface.ProcessStart := FALSE;
            // Action Qualifier=R
            // Token: "ChangeOver_DB".Robot_3.MaintenancePosReqSelFlag
            "ChangeOver_DB".Robot_3.MaintenancePosReqSelFlag := FALSE;
            // Action Qualifier=N
            // Token: //"Robot_DB".Robot_3.MasteringTest_Req
            //"Robot_DB".Robot_3.MasteringTest_Req;
            // Action Qualifier=N
            // Token: //"Robot_DB".Robot_3.BrakeTest_Req
            //"Robot_DB".Robot_3.BrakeTest_Req;
            // Action Qualifier=R
            // Token: #Auto_Run_after_NG_box_closed
            #Auto_Run_after_NG_box_closed := FALSE;

            // Transition to next step: 929
            IF TRUE THEN  // Sequential transition - review XML for actual condition
                #State := STEP_ST10_Flow15_FRobot_3_BrakeTestFinish;
            END_IF;

        // ===========================================
        // STEP 929: BrakeTestFinish
        // ===========================================
        STEP_ST10_Flow15_FRobot_3_BrakeTestFinish:
            // Action Qualifier=R
            // Token: "Robot_DB".Robot_3.BrakeTest_Req
            "Robot_DB".Robot_3.BrakeTest_Req := FALSE;

            // Transition to next step: 373
            IF TRUE THEN  // Sequential transition - review XML for actual condition
                #State := STEP_ST10_Flow15_FRobot_3_StartRobotNG2Put_1;
            END_IF;

        // ===========================================
        // STEP 373: StartRobotNG2Put_1
        // ===========================================
        STEP_ST10_Flow15_FRobot_3_StartRobotNG2Put_1:
            // Action Qualifier=N
            // Token: "KukaRobot3_CtrlDB".sPLCtoROB.User.Cycle.DI266_LoadGlueNGReq2
            "KukaRobot3_CtrlDB".sPLCtoROB.User.Cycle.DI266_LoadGlueNGReq2;

            // Transition to next step: 165
            IF TRUE THEN  // Sequential transition - review XML for actual condition
                #State := STEP_ST10_Flow15_FRobot_3_NG2Put_2_Magnet;
            END_IF;

        // ===========================================
        // STEP 165: NG2Put_2/Magnet
        // ===========================================
        STEP_ST10_Flow15_FRobot_3_NG2Put_2_Magnet:
            // Action Qualifier=R
            // Token: #ioPM_Inface.ProcessComplete
            #ioPM_Inface.ProcessComplete := FALSE;
            // Action Qualifier=S
            // Token: #ioPM_Inface.ProcessStart
            #ioPM_Inface.ProcessStart := TRUE;

            // Transition to next step: 319
            IF TRUE THEN  // Sequential transition - review XML for actual condition
                #State := STEP_ST10_Flow15_FRobot_3_WaitPos4ScanFinish;
            END_IF;

        // ===========================================
        // STEP 319: WaitPos4ScanFinish
        // ===========================================
        STEP_ST10_Flow15_FRobot_3_WaitPos4ScanFinish:
            // No actions in XML

            // Transition to next step: 273
            IF TRUE THEN  // Sequential transition - review XML for actual condition
                #State := STEP_ST10_Flow15_FRobot_3_PartOKStatus_1;
            END_IF;

        // ===========================================
        // STEP 273: PartOKStatus_1
        // ===========================================
        STEP_ST10_Flow15_FRobot_3_PartOKStatus_1:
            // Action Qualifier=N
            // Token: "AutoProcessData".F_Robot3Grip2.PartStatus := 110
            "AutoProcessData".F_Robot3Grip2.PartStatus := 110;

            // Transition to next step: 899
            IF TRUE THEN  // Sequential transition - review XML for actual condition
                #State := STEP_ST10_Flow15_FRobot_3_WaitR1HomePosFinsh_1;
            END_IF;

        // ===========================================
        // STEP 899: WaitR1HomePosFinsh_1
        // ===========================================
        STEP_ST10_Flow15_FRobot_3_WaitR1HomePosFinsh_1:
            // Action Qualifier=R
            // Token: "AutoProcessControl".Robot_3.HomeRequest
            "AutoProcessControl".Robot_3.HomeRequest := FALSE;

            // Transition to next step: 337
            IF TRUE THEN  // Sequential transition - review XML for actual condition
                #State := STEP_ST10_Flow15_FRobot_3_RobotScanGripperReachPos2;
            END_IF;

        // ===========================================
        // STEP 337: RobotScanGripperReachPos2
        // ===========================================
        STEP_ST10_Flow15_FRobot_3_RobotScanGripperReachPos2:
            // No actions in XML

            // Transition to next step: 328
            IF TRUE THEN  // Sequential transition - review XML for actual condition
                #State := STEP_ST10_Flow15_FRobot_3_StartRobotPickGlueNG;
            END_IF;

        // ===========================================
        // STEP 328: StartRobotPickGlueNG
        // ===========================================
        STEP_ST10_Flow15_FRobot_3_StartRobotPickGlueNG:
            // Action Qualifier=N
            // Token: "KukaRobot3_CtrlDB".sPLCtoROB.User.Cycle.DI253_PickGlueNGReq
            "KukaRobot3_CtrlDB".sPLCtoROB.User.Cycle.DI253_PickGlueNGReq;

            // Transition to next step: 599
            IF TRUE THEN  // Sequential transition - review XML for actual condition
                #State := STEP_ST10_Flow15_FRobot_3_PressRingPutProcessFinish;
            END_IF;

        // ===========================================
        // STEP 599: PressRingPutProcessFinish
        // ===========================================
        STEP_ST10_Flow15_FRobot_3_PressRingPutProcessFinish:
            // Action Qualifier=S
            // Token: #ioPM_Inface.ProcessComplete
            #ioPM_Inface.ProcessComplete := TRUE;
            // Action Qualifier=R
            // Token: #ioPM_Inface.ProcessStart
            #ioPM_Inface.ProcessStart := FALSE;

            // Transition to next step: 334
            IF TRUE THEN  // Sequential transition - review XML for actual condition
                #State := STEP_ST10_Flow15_FRobot_3_StartRobotScanGripperCode;
            END_IF;

        // ===========================================
        // STEP 334: StartRobotScanGripperCode
        // ===========================================
        STEP_ST10_Flow15_FRobot_3_StartRobotScanGripperCode:
            // Action Qualifier=N
            // Token: "KukaRobot3_CtrlDB".sPLCtoROB.User.Cycle.DI305_GripScan
            "KukaRobot3_CtrlDB".sPLCtoROB.User.Cycle.DI305_GripScan;

            // Transition to next step: 270
            IF TRUE THEN  // Sequential transition - review XML for actual condition
                #State := STEP_ST10_Flow15_FRobot_3_DataMove_7;
            END_IF;

        // ===========================================
        // STEP 270: DataMove_7
        // ===========================================
        STEP_ST10_Flow15_FRobot_3_DataMove_7:
            // Action Qualifier=N
            // Token: //"AutoProcessData_Buffer".DataBuffer["AutoProcessData".GlobalData.DataIndex]:="AutoProcessData".F_Robot3Grip2
            //"AutoProcessData_Buffer".DataBuffer["AutoProcessData".GlobalData.DataIndex]:="AutoProcessData".F_Robot3Grip2;
            // Action Qualifier=N
            // Token: //"AutoProcessData".GlobalData.DataIndex:="AutoProcessData".GlobalData.DataIndex+1
            //"AutoProcessData".GlobalData.DataIndex:="AutoProcessData".GlobalData.DataIndex+1;

            // Transition to next step: 131
            IF TRUE THEN  // Sequential transition - review XML for actual condition
                #State := STEP_ST10_Flow15_FRobot_3_Maintenance;
            END_IF;

        // ===========================================
        // STEP 131: Maintenance
        // ===========================================
        STEP_ST10_Flow15_FRobot_3_Maintenance:
            // Action Qualifier=R
            // Token: #ioPM_Inface.ProcessComplete
            #ioPM_Inface.ProcessComplete := FALSE;
            // Action Qualifier=S
            // Token: #ioPM_Inface.ProcessStart
            #ioPM_Inface.ProcessStart := TRUE;

            // Transition to next step: 243
            IF TRUE THEN  // Sequential transition - review XML for actual condition
                #State := STEP_ST10_Flow15_FRobot_3_Grip1PartStatus;
            END_IF;

        // ===========================================
        // STEP 243: Grip1PartStatus
        // ===========================================
        STEP_ST10_Flow15_FRobot_3_Grip1PartStatus:
            // Action Qualifier=N
            // Token: "AutoProcessData".F_Robot3Grip1.PartStatus := 100
            "AutoProcessData".F_Robot3Grip1.PartStatus := 100;

            // Transition to next step: 381
            IF TRUE THEN  // Sequential transition - review XML for actual condition
                #State := STEP_ST10_Flow15_FRobot_3_Grip1SensorError;
            END_IF;

        // ===========================================
        // STEP 381: Grip1SensorError
        // ===========================================
        STEP_ST10_Flow15_FRobot_3_Grip1SensorError:
            // Action Qualifier=S
            // Token: "ST10_DeviceError".F.Robot_3.Grip1SensorCheckError
            "ST10_DeviceError".F.Robot_3.Grip1SensorCheckError := TRUE;

            // Transition to next step: 911
            IF TRUE THEN  // Sequential transition - review XML for actual condition
                #State := STEP_ST10_Flow15_FRobot_3_WaitMasteringTestFinish;
            END_IF;

        // ===========================================
        // STEP 911: WaitMasteringTestFinish
        // ===========================================
        STEP_ST10_Flow15_FRobot_3_WaitMasteringTestFinish:
            // No actions in XML

            // Transition to next step: 262
            IF TRUE THEN  // Sequential transition - review XML for actual condition
                #State := STEP_ST10_Flow15_FRobot_3_DataMove_4;
            END_IF;

        // ===========================================
        // STEP 262: DataMove_4
        // ===========================================
        STEP_ST10_Flow15_FRobot_3_DataMove_4:
            // Action Qualifier=N, Event="S1"
            // Token: "AutoProcessData".F_Robot3Grip1 := "AutoProcessData".B_Press2
            "AutoProcessData".F_Robot3Grip1 := "AutoProcessData".B_Press2;
            // Action Qualifier=N, Event="S1"
            // Token: "AutoProcessData".B_Press2 := "AutoProcessData".ClearData
            "AutoProcessData".B_Press2 := "AutoProcessData".ClearData;

            // Transition to next step: 140
            IF TRUE THEN  // Sequential transition - review XML for actual condition
                #State := STEP_ST10_Flow15_FRobot_3_PressShaftPut;
            END_IF;

        // ===========================================
        // STEP 140: PressShaftPut
        // ===========================================
        STEP_ST10_Flow15_FRobot_3_PressShaftPut:
            // Action Qualifier=R
            // Token: #ioPM_Inface.ProcessComplete
            #ioPM_Inface.ProcessComplete := FALSE;
            // Action Qualifier=S
            // Token: #ioPM_Inface.ProcessStart
            #ioPM_Inface.ProcessStart := TRUE;

            // Transition to next step: 359
            IF TRUE THEN  // Sequential transition - review XML for actual condition
                #State := STEP_ST10_Flow15_FRobot_3_WaitRobotFinish_5;
            END_IF;

        // ===========================================
        // STEP 359: WaitRobotFinish_5
        // ===========================================
        STEP_ST10_Flow15_FRobot_3_WaitRobotFinish_5:
            // No actions in XML

            // Transition to next step: 346
            IF TRUE THEN  // Sequential transition - review XML for actual condition
                #State := STEP_ST10_Flow15_FRobot_3_WaitRobotGripHaveStatus;
            END_IF;

        // ===========================================
        // STEP 346: WaitRobotGripHaveStatus
        // ===========================================
        STEP_ST10_Flow15_FRobot_3_WaitRobotGripHaveStatus:
            // No actions in XML

            // Transition to next step: 343
            IF TRUE THEN  // Sequential transition - review XML for actual condition
                #State := STEP_ST10_Flow15_FRobot_3_WaitRobotFinish_1;
            END_IF;

        // ===========================================
        // STEP 343: WaitRobotFinish_1
        // ===========================================
        STEP_ST10_Flow15_FRobot_3_WaitRobotFinish_1:
            // No actions in XML

            // Transition to next step: 336
            IF TRUE THEN  // Sequential transition - review XML for actual condition
                #State := STEP_ST10_Flow15_FRobot_3_WaitGripperPos1ScanFinish;
            END_IF;

        // ===========================================
        // STEP 336: WaitGripperPos1ScanFinish
        // ===========================================
        STEP_ST10_Flow15_FRobot_3_WaitGripperPos1ScanFinish:
            // No actions in XML

            // Transition to next step: 316
            IF TRUE THEN  // Sequential transition - review XML for actual condition
                #State := STEP_ST10_Flow15_FRobot_3_RobotStart;
            END_IF;

        // ===========================================
        // STEP 316: RobotStart
        // ===========================================
        STEP_ST10_Flow15_FRobot_3_RobotStart:
            // Action Qualifier=N
            // Token: "KukaRobot3_CtrlDB".ioAutoStart
            "KukaRobot3_CtrlDB".ioAutoStart;

            // Transition to next step: 312
            IF TRUE THEN  // Sequential transition - review XML for actual condition
                #State := STEP_ST10_Flow15_FRobot_3_WaitPos2ScanFinish;
            END_IF;

        // ===========================================
        // STEP 312: WaitPos2ScanFinish
        // ===========================================
        STEP_ST10_Flow15_FRobot_3_WaitPos2ScanFinish:
            // No actions in XML

            // Transition to next step: 313
            IF TRUE THEN  // Sequential transition - review XML for actual condition
                #State := STEP_ST10_Flow15_FRobot_3_WaitRobotReachPos2;
            END_IF;

        // ===========================================
        // STEP 313: WaitRobotReachPos2
        // ===========================================
        STEP_ST10_Flow15_FRobot_3_WaitRobotReachPos2:
            // No actions in XML

            // Transition to next step: 317
            IF TRUE THEN  // Sequential transition - review XML for actual condition
                #State := STEP_ST10_Flow15_FRobot_3_RobotHome;
            END_IF;

        // ===========================================
        // STEP 317: RobotHome
        // ===========================================
        STEP_ST10_Flow15_FRobot_3_RobotHome:
            // Action Qualifier=N
            // Token: "KukaRobot3_CtrlDB".ioSrartHome
            "KukaRobot3_CtrlDB".ioSrartHome;

            // Transition to next step: 342
            IF TRUE THEN  // Sequential transition - review XML for actual condition
                #State := STEP_ST10_Flow15_FRobot_3_WaitGripperPos4ScanFinish;
            END_IF;

        // ===========================================
        // STEP 342: WaitGripperPos4ScanFinish
        // ===========================================
        STEP_ST10_Flow15_FRobot_3_WaitGripperPos4ScanFinish:
            // No actions in XML

            // Transition to next step: 247
            IF TRUE THEN  // Sequential transition - review XML for actual condition
                #State := STEP_ST10_Flow15_FRobot_3_WaitScanCompletely;
            END_IF;

        // ===========================================
        // STEP 247: WaitScanCompletely
        // ===========================================
        STEP_ST10_Flow15_FRobot_3_WaitScanCompletely:
            // No actions in XML

            // Transition to next step: 349
            IF TRUE THEN  // Sequential transition - review XML for actual condition
                #State := STEP_ST10_Flow15_FRobot_3_PickGlueNGFinish_1;
            END_IF;

        // ===========================================
        // STEP 349: PickGlueNGFinish_1
        // ===========================================
        STEP_ST10_Flow15_FRobot_3_PickGlueNGFinish_1:
            // Action Qualifier=S
            // Token: #ioPM_Inface.ProcessComplete
            #ioPM_Inface.ProcessComplete := TRUE;
            // Action Qualifier=R
            // Token: #ioPM_Inface.ProcessStart
            #ioPM_Inface.ProcessStart := FALSE;

            // Transition to next step: 244
            IF TRUE THEN  // Sequential transition - review XML for actual condition
                #State := STEP_ST10_Flow15_FRobot_3_Grip2PartStatus;
            END_IF;

        // ===========================================
        // STEP 244: Grip2PartStatus
        // ===========================================
        STEP_ST10_Flow15_FRobot_3_Grip2PartStatus:
            // Action Qualifier=N
            // Token: "AutoProcessData".F_Robot3Grip2.PartStatus := 100
            "AutoProcessData".F_Robot3Grip2.PartStatus := 100;

            // Transition to next step: 353
            IF TRUE THEN  // Sequential transition - review XML for actual condition
                #State := STEP_ST10_Flow15_FRobot_3_WaitRobotFinish_3;
            END_IF;

        // ===========================================
        // STEP 353: WaitRobotFinish_3
        // ===========================================
        STEP_ST10_Flow15_FRobot_3_WaitRobotFinish_3:
            // No actions in XML

            // Transition to next step: 363
            IF TRUE THEN  // Sequential transition - review XML for actual condition
                #State := STEP_ST10_Flow15_FRobot_3_WaitRobotGripStatus_1;
            END_IF;

        // ===========================================
        // STEP 363: WaitRobotGripStatus_1
        // ===========================================
        STEP_ST10_Flow15_FRobot_3_WaitRobotGripStatus_1:
            // No actions in XML

            // Transition to next step: 170
            IF TRUE THEN  // Sequential transition - review XML for actual condition
                #State := STEP_ST10_Flow15_FRobot_3_NG2Put_3_Ring;
            END_IF;

        // ===========================================
        // STEP 170: NG2Put_3/Ring
        // ===========================================
        STEP_ST10_Flow15_FRobot_3_NG2Put_3_Ring:
            // Action Qualifier=R
            // Token: #ioPM_Inface.ProcessComplete
            #ioPM_Inface.ProcessComplete := FALSE;
            // Action Qualifier=S
            // Token: #ioPM_Inface.ProcessStart
            #ioPM_Inface.ProcessStart := TRUE;

            // Transition to next step: 272
            IF TRUE THEN  // Sequential transition - review XML for actual condition
                #State := STEP_ST10_Flow15_FRobot_3_FlagReset;
            END_IF;

        // ===========================================
        // STEP 272: FlagReset
        // ===========================================
        STEP_ST10_Flow15_FRobot_3_FlagReset:
            // Action Qualifier=R
            // Token: "AutoProcessControl".Robot_3.Press2PutFlag
            "AutoProcessControl".Robot_3.Press2PutFlag := FALSE;
            // Action Qualifier=R
            // Token: "AutoProcessControl".Robot_3.Press2PickFlag
            "AutoProcessControl".Robot_3.Press2PickFlag := FALSE;
            // Action Qualifier=R
            // Token: "AutoProcessControl".Robot_3.GlueNGPickFlag
            "AutoProcessControl".Robot_3.GlueNGPickFlag := FALSE;
            // Action Qualifier=R
            // Token: "AutoProcessControl".Robot_3.ScanNGPickFlag
            "AutoProcessControl".Robot_3.ScanNGPickFlag := FALSE;
            // Action Qualifier=R
            // Token: "AutoProcessControl".Robot_3.NGPutFlag
            "AutoProcessControl".Robot_3.NGPutFlag := FALSE;

            // Transition to next step: 366
            IF TRUE THEN  // Sequential transition - review XML for actual condition
                #State := STEP_ST10_Flow15_FRobot_3_WaitRobotGripStatus_2;
            END_IF;

        // ===========================================
        // STEP 366: WaitRobotGripStatus_2
        // ===========================================
        STEP_ST10_Flow15_FRobot_3_WaitRobotGripStatus_2:
            // No actions in XML

            // Transition to next step: 362
            IF TRUE THEN  // Sequential transition - review XML for actual condition
                #State := STEP_ST10_Flow15_FRobot_3_WaitRobotFinish_6;
            END_IF;

        // ===========================================
        // STEP 362: WaitRobotFinish_6
        // ===========================================
        STEP_ST10_Flow15_FRobot_3_WaitRobotFinish_6:
            // No actions in XML

            // Transition to next step: 332
            IF TRUE THEN  // Sequential transition - review XML for actual condition
                #State := STEP_ST10_Flow15_FRobot_3_Gripe2StatusAlarm;
            END_IF;

        // ===========================================
        // STEP 332: Gripe2StatusAlarm
        // ===========================================
        STEP_ST10_Flow15_FRobot_3_Gripe2StatusAlarm:
            // Action Qualifier=S
            // Token: "ST10_DeviceError".F.Robot_3.Grip2Error
            "ST10_DeviceError".F.Robot_3.Grip2Error := TRUE;

            // Transition to next step: 271
            IF TRUE THEN  // Sequential transition - review XML for actual condition
                #State := STEP_ST10_Flow15_FRobot_3_DataMove_8;
            END_IF;

        // ===========================================
        // STEP 271: DataMove_8
        // ===========================================
        STEP_ST10_Flow15_FRobot_3_DataMove_8:
            // Action Qualifier=N
            // Token: //"AutoProcessData_Buffer".DataBuffer["AutoProcessData".GlobalData.DataIndex]:="AutoProcessData".F_Robot3Grip2
            //"AutoProcessData_Buffer".DataBuffer["AutoProcessData".GlobalData.DataIndex]:="AutoProcessData".F_Robot3Grip2;
            // Action Qualifier=N
            // Token: //"AutoProcessData".GlobalData.DataIndex:="AutoProcessData".GlobalData.DataIndex+1
            //"AutoProcessData".GlobalData.DataIndex:="AutoProcessData".GlobalData.DataIndex+1;

            // Transition to next step: 352
            IF TRUE THEN  // Sequential transition - review XML for actual condition
                #State := STEP_ST10_Flow15_FRobot_3_StartRobotPickTable;
            END_IF;

        // ===========================================
        // STEP 352: StartRobotPickTable
        // ===========================================
        STEP_ST10_Flow15_FRobot_3_StartRobotPickTable:
            // Action Qualifier=N
            // Token: "KukaRobot3_CtrlDB".sPLCtoROB.User.Cycle.DI257_PickTableReq
            "KukaRobot3_CtrlDB".sPLCtoROB.User.Cycle.DI257_PickTableReq;

            // Transition to next step: 246
            IF TRUE THEN  // Sequential transition - review XML for actual condition
                #State := STEP_ST10_Flow15_FRobot_3_ScanStart;
            END_IF;

        // ===========================================
        // STEP 246: ScanStart
        // ===========================================
        STEP_ST10_Flow15_FRobot_3_ScanStart:
            // Action Qualifier=S
            // Token: "KeyenceSR1000Ctrl_803A1DB".ioAutoTrigger
            "KeyenceSR1000Ctrl_803A1DB".ioAutoTrigger := TRUE;

            // Transition to next step: 120
            IF TRUE THEN  // Sequential transition - review XML for actual condition
                #State := STEP_ST10_Flow15_FRobot_3_PickGlueNGReq;
            END_IF;

        // ===========================================
        // STEP 120: PickGlueNGReq
        // ===========================================
        STEP_ST10_Flow15_FRobot_3_PickGlueNGReq:
            // Action Qualifier=R
            // Token: #ioPM_Inface.ProcessComplete
            #ioPM_Inface.ProcessComplete := FALSE;
            // Action Qualifier=S
            // Token: #ioPM_Inface.ProcessStart
            #ioPM_Inface.ProcessStart := TRUE;

            // Transition to next step: 4
            IF TRUE THEN  // Sequential transition - review XML for actual condition
                #State := STEP_ST10_Flow15_FRobot_3_RobotSpeed;
            END_IF;

        // ===========================================
        // STEP 4: RobotSpeed
        // ===========================================
        STEP_ST10_Flow15_FRobot_3_RobotSpeed:
            // Action Qualifier=N
            // Token: "KukaRobot3_CtrlDB".iSpeedValue := 20
            "KukaRobot3_CtrlDB".iSpeedValue := 20;

            // Transition to next step: 364
            IF TRUE THEN  // Sequential transition - review XML for actual condition
                #State := STEP_ST10_Flow15_FRobot_3_StartRobotPressPick;
            END_IF;

        // ===========================================
        // STEP 364: StartRobotPressPick
        // ===========================================
        STEP_ST10_Flow15_FRobot_3_StartRobotPressPick:
            // Action Qualifier=N
            // Token: "KukaRobot3_CtrlDB".sPLCtoROB.User.Cycle.DI281_PressPickPartReq
            "KukaRobot3_CtrlDB".sPLCtoROB.User.Cycle.DI281_PressPickPartReq;

            // Transition to next step: 385
            IF TRUE THEN  // Sequential transition - review XML for actual condition
                #State := STEP_ST10_Flow15_FRobot_3_MES_Online__offline_;
            END_IF;

        // ===========================================
        // STEP 385: MES Online  offline?
        // ===========================================
        STEP_ST10_Flow15_FRobot_3_MES_Online__offline_:
            // No actions in XML

            // Transition to next step: 10
            IF TRUE THEN  // Sequential transition - review XML for actual condition
                #State := STEP_ST10_Flow15_FRobot_3_S10_InitialFinish;
            END_IF;

        // ===========================================
        // STEP 10: S10_InitialFinish
        // ===========================================
        STEP_ST10_Flow15_FRobot_3_S10_InitialFinish:
            // Action Qualifier=S
            // Token: #ioPM_Inface.InitialOK
            #ioPM_Inface.InitialOK := TRUE;

            // Transition to next step: 399
            IF TRUE THEN  // Sequential transition - review XML for actual condition
                #State := STEP_ST10_Flow15_FRobot_3_PickMagnScanNGBufferFinish;
            END_IF;

        // ===========================================
        // STEP 399: PickMagnScanNGBufferFinish
        // ===========================================
        STEP_ST10_Flow15_FRobot_3_PickMagnScanNGBufferFinish:
            // Action Qualifier=S
            // Token: #ioPM_Inface.ProcessComplete
            #ioPM_Inface.ProcessComplete := TRUE;
            // Action Qualifier=R
            // Token: #ioPM_Inface.ProcessStart
            #ioPM_Inface.ProcessStart := FALSE;

            // Transition to next step: 339
            IF TRUE THEN  // Sequential transition - review XML for actual condition
                #State := STEP_ST10_Flow15_FRobot_3_RobotScanGripperReachPos3;
            END_IF;

        // ===========================================
        // STEP 339: RobotScanGripperReachPos3
        // ===========================================
        STEP_ST10_Flow15_FRobot_3_RobotScanGripperReachPos3:
            // No actions in XML

            // Transition to next step: 330
            IF TRUE THEN  // Sequential transition - review XML for actual condition
                #State := STEP_ST10_Flow15_FRobot_3_GripStatusCheck;
            END_IF;

        // ===========================================
        // STEP 330: GripStatusCheck
        // ===========================================
        STEP_ST10_Flow15_FRobot_3_GripStatusCheck:
            // No actions in XML

            // Transition to next step: 450
            IF TRUE THEN  // Sequential transition - review XML for actual condition
                #State := STEP_ST10_Flow15_FRobot_3_ScanRingProcess;
            END_IF;

        // ===========================================
        // STEP 450: ScanRingProcess
        // ===========================================
        STEP_ST10_Flow15_FRobot_3_ScanRingProcess:
            // No actions in XML

            // Transition to next step: 3
            IF TRUE THEN  // Sequential transition - review XML for actual condition
                #State := STEP_ST10_Flow15_FRobot_3_S3;
            END_IF;

        // ===========================================
        // STEP 3: S3
        // ===========================================
        STEP_ST10_Flow15_FRobot_3_S3:
            // No actions in XML

            // Transition to next step: 750
            IF TRUE THEN  // Sequential transition - review XML for actual condition
                #State := STEP_ST10_Flow15_FRobot_3_NG_2_PutProcess;
            END_IF;

        // ===========================================
        // STEP 750: NG 2 PutProcess
        // ===========================================
        STEP_ST10_Flow15_FRobot_3_NG_2_PutProcess:
            // No actions in XML

            // Transition to next step: 374
            IF TRUE THEN  // Sequential transition - review XML for actual condition
                #State := STEP_ST10_Flow15_FRobot_3_WaitRobotFinish_10;
            END_IF;

        // ===========================================
        // STEP 374: WaitRobotFinish_10
        // ===========================================
        STEP_ST10_Flow15_FRobot_3_WaitRobotFinish_10:
            // No actions in XML

            // Transition to next step: 650
            IF TRUE THEN  // Sequential transition - review XML for actual condition
                #State := STEP_ST10_Flow15_FRobot_3_GluePutProcess;
            END_IF;

        // ===========================================
        // STEP 650: GluePutProcess
        // ===========================================
        STEP_ST10_Flow15_FRobot_3_GluePutProcess:
            // No actions in XML

            // Transition to next step: 449
            IF TRUE THEN  // Sequential transition - review XML for actual condition
                #State := STEP_ST10_Flow15_FRobot_3_PickTableProcessFinish;
            END_IF;

        // ===========================================
        // STEP 449: PickTableProcessFinish
        // ===========================================
        STEP_ST10_Flow15_FRobot_3_PickTableProcessFinish:
            // Action Qualifier=S
            // Token: #ioPM_Inface.ProcessComplete
            #ioPM_Inface.ProcessComplete := TRUE;
            // Action Qualifier=R
            // Token: #ioPM_Inface.ProcessStart
            #ioPM_Inface.ProcessStart := FALSE;

            // Transition to next step: 252
            IF TRUE THEN  // Sequential transition - review XML for actual condition
                #State := STEP_ST10_Flow15_FRobot_3_DataClear;
            END_IF;

        // ===========================================
        // STEP 252: DataClear
        // ===========================================
        STEP_ST10_Flow15_FRobot_3_DataClear:
            // Action Qualifier=N, Event="S1"
            // Token: "AutoProcessData".F_Robot3Grip1 := "AutoProcessData".ClearData
            "AutoProcessData".F_Robot3Grip1 := "AutoProcessData".ClearData;

            // Transition to next step: 258
            IF TRUE THEN  // Sequential transition - review XML for actual condition
                #State := STEP_ST10_Flow15_FRobot_3_Data_Clear_2;
            END_IF;

        // ===========================================
        // STEP 258: Data Clear_2
        // ===========================================
        STEP_ST10_Flow15_FRobot_3_Data_Clear_2:
            // Action Qualifier=N, Event="S1"
            // Token: "AutoProcessData".F_Robot3Grip2 := "AutoProcessData".ClearData
            "AutoProcessData".F_Robot3Grip2 := "AutoProcessData".ClearData;

            // Transition to next step: 125
            IF TRUE THEN  // Sequential transition - review XML for actual condition
                #State := STEP_ST10_Flow15_FRobot_3_PickMagnetNGReqPick;
            END_IF;

        // ===========================================
        // STEP 125: PickMagnetNGReqPick
        // ===========================================
        STEP_ST10_Flow15_FRobot_3_PickMagnetNGReqPick:
            // Action Qualifier=R
            // Token: #ioPM_Inface.ProcessComplete
            #ioPM_Inface.ProcessComplete := FALSE;
            // Action Qualifier=S
            // Token: #ioPM_Inface.ProcessStart
            #ioPM_Inface.ProcessStart := TRUE;
            // Action Qualifier=S
            // Token: "AutoProcessControl".Robot_3.ScanNGPickFlag
            "AutoProcessControl".Robot_3.ScanNGPickFlag := TRUE;

            // Transition to next step: 550
            IF TRUE THEN  // Sequential transition - review XML for actual condition
                #State := STEP_ST10_Flow15_FRobot_3_PressRingPutProcess;
            END_IF;

        // ===========================================
        // STEP 550: PressRingPutProcess
        // ===========================================
        STEP_ST10_Flow15_FRobot_3_PressRingPutProcess:
            // No actions in XML

            // Transition to next step: 345
            IF TRUE THEN  // Sequential transition - review XML for actual condition
                #State := STEP_ST10_Flow15_FRobot_3_WaitRobotFinish_2;
            END_IF;

        // ===========================================
        // STEP 345: WaitRobotFinish_2
        // ===========================================
        STEP_ST10_Flow15_FRobot_3_WaitRobotFinish_2:
            // No actions in XML

            // Transition to next step: 400
            IF TRUE THEN  // Sequential transition - review XML for actual condition
                #State := STEP_ST10_Flow15_FRobot_3_PickTableProcess;
            END_IF;

        // ===========================================
        // STEP 400: PickTableProcess
        // ===========================================
        STEP_ST10_Flow15_FRobot_3_PickTableProcess:
            // No actions in XML

            // Transition to next step: 354
            IF TRUE THEN  // Sequential transition - review XML for actual condition
                #State := STEP_ST10_Flow15_FRobot_3_WaitRobotGripHaveStatus_3;
            END_IF;

        // ===========================================
        // STEP 354: WaitRobotGripHaveStatus_3
        // ===========================================
        STEP_ST10_Flow15_FRobot_3_WaitRobotGripHaveStatus_3:
            // No actions in XML

            // Transition to next step: 700
            IF TRUE THEN  // Sequential transition - review XML for actual condition
                #State := STEP_ST10_Flow15_FRobot_3_NG_PutProcess;
            END_IF;

        // ===========================================
        // STEP 700: NG PutProcess
        // ===========================================
        STEP_ST10_Flow15_FRobot_3_NG_PutProcess:
            // No actions in XML

            // Transition to next step: 370
            IF TRUE THEN  // Sequential transition - review XML for actual condition
                #State := STEP_ST10_Flow15_FRobot_3_StartRobotNGPut;
            END_IF;

        // ===========================================
        // STEP 370: StartRobotNGPut
        // ===========================================
        STEP_ST10_Flow15_FRobot_3_StartRobotNGPut:
            // Action Qualifier=N
            // Token: "KukaRobot3_CtrlDB".sPLCtoROB.User.Cycle.DI265_LoadPressNGReq1
            "KukaRobot3_CtrlDB".sPLCtoROB.User.Cycle.DI265_LoadPressNGReq1;

            // Transition to next step: 314
            IF TRUE THEN  // Sequential transition - review XML for actual condition
                #State := STEP_ST10_Flow15_FRobot_3_WaitRobotReachPos3;
            END_IF;

        // ===========================================
        // STEP 314: WaitRobotReachPos3
        // ===========================================
        STEP_ST10_Flow15_FRobot_3_WaitRobotReachPos3:
            // No actions in XML

            // Transition to next step: 850
            IF TRUE THEN  // Sequential transition - review XML for actual condition
                #State := STEP_ST10_Flow15_FRobot_3_Maintenance_Pos;
            END_IF;

        // ===========================================
        // STEP 850: Maintenance Pos
        // ===========================================
        STEP_ST10_Flow15_FRobot_3_Maintenance_Pos:
            // No actions in XML

            // Transition to next step: 600
            IF TRUE THEN  // Sequential transition - review XML for actual condition
                #State := STEP_ST10_Flow15_FRobot_3_PressPickProcess;
            END_IF;

        // ===========================================
        // STEP 600: PressPickProcess
        // ===========================================
        STEP_ST10_Flow15_FRobot_3_PressPickProcess:
            // No actions in XML

            // Transition to next step: 269
            IF TRUE THEN  // Sequential transition - review XML for actual condition
                #State := STEP_ST10_Flow15_FRobot_3_Data_Clear_9;
            END_IF;

        // ===========================================
        // STEP 269: Data Clear_9
        // ===========================================
        STEP_ST10_Flow15_FRobot_3_Data_Clear_9:
            // Action Qualifier=N
            // Token: "AutoProcessData".F_Robot3Grip2 := "AutoProcessData".ClearData
            "AutoProcessData".F_Robot3Grip2 := "AutoProcessData".ClearData;

            // Transition to next step: 649
            IF TRUE THEN  // Sequential transition - review XML for actual condition
                #State := STEP_ST10_Flow15_FRobot_3_PressPickProcessFinish_;
            END_IF;

        // ===========================================
        // STEP 649: PressPickProcessFinish_
        // ===========================================
        STEP_ST10_Flow15_FRobot_3_PressPickProcessFinish_:
            // Action Qualifier=S
            // Token: #ioPM_Inface.ProcessComplete
            #ioPM_Inface.ProcessComplete := TRUE;
            // Action Qualifier=R
            // Token: #ioPM_Inface.ProcessStart
            #ioPM_Inface.ProcessStart := FALSE;

            // Transition to next step: 338
            IF TRUE THEN  // Sequential transition - review XML for actual condition
                #State := STEP_ST10_Flow15_FRobot_3_WaitGripperPos2ScanFinish;
            END_IF;

        // ===========================================
        // STEP 338: WaitGripperPos2ScanFinish
        // ===========================================
        STEP_ST10_Flow15_FRobot_3_WaitGripperPos2ScanFinish:
            // No actions in XML

            // Transition to next step: 200
            IF TRUE THEN  // Sequential transition - review XML for actual condition
                #State := STEP_ST10_Flow15_FRobot_3_Tablecode_Scan;
            END_IF;

        // ===========================================
        // STEP 200: Tablecode Scan
        // ===========================================
        STEP_ST10_Flow15_FRobot_3_Tablecode_Scan:
            // No actions in XML

            // Transition to next step: 910
            IF TRUE THEN  // Sequential transition - review XML for actual condition
                #State := STEP_ST10_Flow15_FRobot_3_MasteringTest_Req;
            END_IF;

        // ===========================================
        // STEP 910: MasteringTest_Req
        // ===========================================
        STEP_ST10_Flow15_FRobot_3_MasteringTest_Req:
            // Action Qualifier=N
            // Token: "KukaRobot3_CtrlDB".sPLCtoROB.User.Cycle.DI321
            "KukaRobot3_CtrlDB".sPLCtoROB.User.Cycle.DI321;
            // Action Qualifier=N
            // Token: "KukaRobot3_CtrlDB".sPLCtoROB.User.Safety.DI450
            "KukaRobot3_CtrlDB".sPLCtoROB.User.Safety.DI450;

            // Transition to next step: 100
            IF TRUE THEN  // Sequential transition - review XML for actual condition
                #State := STEP_ST10_Flow15_FRobot_3_ProcessStart;
            END_IF;

        // ===========================================
        // STEP 100: ProcessStart
        // ===========================================
        STEP_ST10_Flow15_FRobot_3_ProcessStart:
            // Action Qualifier=R
            // Token: #ioPM_Inface.InitialRun
            #ioPM_Inface.InitialRun := FALSE;
            // Action Qualifier=R
            // Token: #ioPM_Inface.ProcessComplete
            #ioPM_Inface.ProcessComplete := FALSE;
            // Action Qualifier=R
            // Token: #ioPM_Inface.ProcessStart
            #ioPM_Inface.ProcessStart := FALSE;
            // Action Qualifier=S
            // Token: #ioPM_Inface.InitialOK
            #ioPM_Inface.InitialOK := TRUE;
            // Action Qualifier=S
            // Token: #ioPM_Inface.WaitRunning
            #ioPM_Inface.WaitRunning := TRUE;
            // Action Qualifier=N, Event="S1"
            // Token: #ioPM_Inface.ProcessResult := 0
            #ioPM_Inface.ProcessResult := 0;
            // Action Qualifier=R
            // Token: "ST10_GeneralData".FlowControl_Handshake[5].Start
            "ST10_GeneralData".FlowControl_Handshake[5].Start := FALSE;
            // Action Qualifier=R
            // Token: "ST10_GeneralData".FlowControl_Handshake[5].Done
            "ST10_GeneralData".FlowControl_Handshake[5].Done := FALSE;

            // Transition to next step: 251
            IF TRUE THEN  // Sequential transition - review XML for actual condition
                #State := STEP_ST10_Flow15_FRobot_3_PartNGStatus;
            END_IF;

        // ===========================================
        // STEP 251: PartNGStatus
        // ===========================================
        STEP_ST10_Flow15_FRobot_3_PartNGStatus:
            // Action Qualifier=N
            // Token: "AutoProcessData".F_Robot3Grip2.PartStatus := 150
            "AutoProcessData".F_Robot3Grip2.PartStatus := 150;

            // Transition to next step: 268
            IF TRUE THEN  // Sequential transition - review XML for actual condition
                #State := STEP_ST10_Flow15_FRobot_3_Data_Clear_8;
            END_IF;

        // ===========================================
        // STEP 268: Data Clear_8
        // ===========================================
        STEP_ST10_Flow15_FRobot_3_Data_Clear_8:
            // Action Qualifier=N
            // Token: "AutoProcessData".F_Robot3Grip2 := "AutoProcessData".ClearData
            "AutoProcessData".F_Robot3Grip2 := "AutoProcessData".ClearData;

            // Transition to next step: 384
            IF TRUE THEN  // Sequential transition - review XML for actual condition
                #State := STEP_ST10_Flow15_FRobot_3_RobotManuallyMoved_;
            END_IF;

        // ===========================================
        // STEP 384: RobotManuallyMoved?
        // ===========================================
        STEP_ST10_Flow15_FRobot_3_RobotManuallyMoved_:
            // No actions in XML

            // Transition to next step: 5
            IF TRUE THEN  // Sequential transition - review XML for actual condition
                #State := STEP_ST10_Flow15_FRobot_3_S5_MESInitial;
            END_IF;

        // ===========================================
        // STEP 5: S5_MESInitial
        // ===========================================
        STEP_ST10_Flow15_FRobot_3_S5_MESInitial:
            // No actions in XML

            // Transition to next step: 706
            IF TRUE THEN  // Sequential transition - review XML for actual condition
                #State := STEP_ST10_Flow15_FRobot_3_WaitRobotHomeRequest;
            END_IF;

        // ===========================================
        // STEP 706: WaitRobotHomeRequest
        // ===========================================
        STEP_ST10_Flow15_FRobot_3_WaitRobotHomeRequest:
            // Action Qualifier=R
            // Token: "ChangeOver_DB".Robot_3.MaintenancePosReqSelFlag
            "ChangeOver_DB".Robot_3.MaintenancePosReqSelFlag := FALSE;

            // Transition to next step: 132
            IF TRUE THEN  // Sequential transition - review XML for actual condition
                #State := STEP_ST10_Flow15_FRobot_3_Masref_test;
            END_IF;

        // ===========================================
        // STEP 132: Masref_test
        // ===========================================
        STEP_ST10_Flow15_FRobot_3_Masref_test:
            // Action Qualifier=R
            // Token: #ioPM_Inface.ProcessComplete
            #ioPM_Inface.ProcessComplete := FALSE;
            // Action Qualifier=S
            // Token: #ioPM_Inface.ProcessStart
            #ioPM_Inface.ProcessStart := TRUE;

            // Transition to next step: 920
            IF TRUE THEN  // Sequential transition - review XML for actual condition
                #State := STEP_ST10_Flow15_FRobot_3_BrakeTest_Req;
            END_IF;

        // ===========================================
        // STEP 920: BrakeTest_Req
        // ===========================================
        STEP_ST10_Flow15_FRobot_3_BrakeTest_Req:
            // Action Qualifier=N
            // Token: "KukaRobot3_CtrlDB".sPLCtoROB.User.Cycle.DI329
            "KukaRobot3_CtrlDB".sPLCtoROB.User.Cycle.DI329;
            // Action Qualifier=N
            // Token: "KukaRobot3_CtrlDB".sPLCtoROB.User.Safety.DI451
            "KukaRobot3_CtrlDB".sPLCtoROB.User.Safety.DI451;

            // Transition to next step: 375
            IF TRUE THEN  // Sequential transition - review XML for actual condition
                #State := STEP_ST10_Flow15_FRobot_3_WaitRobotGripStatus_5;
            END_IF;

        // ===========================================
        // STEP 375: WaitRobotGripStatus_5
        // ===========================================
        STEP_ST10_Flow15_FRobot_3_WaitRobotGripStatus_5:
            // No actions in XML

            // Transition to next step: 261
            IF TRUE THEN  // Sequential transition - review XML for actual condition
                #State := STEP_ST10_Flow15_FRobot_3_Data_Clear_4;
            END_IF;

        // ===========================================
        // STEP 261: Data Clear_4
        // ===========================================
        STEP_ST10_Flow15_FRobot_3_Data_Clear_4:
            // Action Qualifier=N, Event="S1"
            // Token: "AutoProcessData".F_Robot3Grip2 := "AutoProcessData".ClearData
            "AutoProcessData".F_Robot3Grip2 := "AutoProcessData".ClearData;

            // Transition to next step: 499
            IF TRUE THEN  // Sequential transition - review XML for actual condition
                #State := STEP_ST10_Flow15_FRobot_3_ScanRingProcessFinish;
            END_IF;

        // ===========================================
        // STEP 499: ScanRingProcessFinish
        // ===========================================
        STEP_ST10_Flow15_FRobot_3_ScanRingProcessFinish:
            // Action Qualifier=S
            // Token: #ioPM_Inface.ProcessComplete
            #ioPM_Inface.ProcessComplete := TRUE;
            // Action Qualifier=R
            // Token: #ioPM_Inface.ProcessStart
            #ioPM_Inface.ProcessStart := FALSE;

            // Transition to next step: 358
            IF TRUE THEN  // Sequential transition - review XML for actual condition
                #State := STEP_ST10_Flow15_FRobot_3_StartRobotPressShaftPut;
            END_IF;

        // ===========================================
        // STEP 358: StartRobotPressShaftPut
        // ===========================================
        STEP_ST10_Flow15_FRobot_3_StartRobotPressShaftPut:
            // Action Qualifier=N
            // Token: "KukaRobot3_CtrlDB".sPLCtoROB.User.Cycle.DI273_PressPutPart1Req
            "KukaRobot3_CtrlDB".sPLCtoROB.User.Cycle.DI273_PressPutPart1Req;

            // Transition to next step: 310
            IF TRUE THEN  // Sequential transition - review XML for actual condition
                #State := STEP_ST10_Flow15_FRobot_3_WaitPos1ScanFinish;
            END_IF;

        // ===========================================
        // STEP 310: WaitPos1ScanFinish
        // ===========================================
        STEP_ST10_Flow15_FRobot_3_WaitPos1ScanFinish:
            // No actions in XML

            // Transition to next step: 308
            IF TRUE THEN  // Sequential transition - review XML for actual condition
                #State := STEP_ST10_Flow15_FRobot_3_StartRobotScanFixtureCode;
            END_IF;

        // ===========================================
        // STEP 308: StartRobotScanFixtureCode
        // ===========================================
        STEP_ST10_Flow15_FRobot_3_StartRobotScanFixtureCode:
            // Action Qualifier=N
            // Token: "KukaRobot3_CtrlDB".sPLCtoROB.User.Cycle.DI225_ScanPosReq
            "KukaRobot3_CtrlDB".sPLCtoROB.User.Cycle.DI225_ScanPosReq;

            // Transition to next step: 344
            IF TRUE THEN  // Sequential transition - review XML for actual condition
                #State := STEP_ST10_Flow15_FRobot_3_StartRobotPickMagnScanNG;
            END_IF;

        // ===========================================
        // STEP 344: StartRobotPickMagnScanNG
        // ===========================================
        STEP_ST10_Flow15_FRobot_3_StartRobotPickMagnScanNG:
            // Action Qualifier=N
            // Token: "KukaRobot3_CtrlDB".sPLCtoROB.User.Cycle.DI249_PickMagnetNGReq
            "KukaRobot3_CtrlDB".sPLCtoROB.User.Cycle.DI249_PickMagnetNGReq;

            // Transition to next step: 110
            IF TRUE THEN  // Sequential transition - review XML for actual condition
                #State := STEP_ST10_Flow15_FRobot_3_ScanFixtureCode;
            END_IF;

        // ===========================================
        // STEP 110: ScanFixtureCode
        // ===========================================
        STEP_ST10_Flow15_FRobot_3_ScanFixtureCode:
            // Action Qualifier=R
            // Token: #ioPM_Inface.ProcessComplete
            #ioPM_Inface.ProcessComplete := FALSE;
            // Action Qualifier=S
            // Token: #ioPM_Inface.ProcessStart
            #ioPM_Inface.ProcessStart := TRUE;

            // Transition to next step: 145
            IF TRUE THEN  // Sequential transition - review XML for actual condition
                #State := STEP_ST10_Flow15_FRobot_3_PressRingPut;
            END_IF;

        // ===========================================
        // STEP 145: PressRingPut
        // ===========================================
        STEP_ST10_Flow15_FRobot_3_PressRingPut:
            // Action Qualifier=R
            // Token: #ioPM_Inface.ProcessComplete
            #ioPM_Inface.ProcessComplete := FALSE;
            // Action Qualifier=S
            // Token: #ioPM_Inface.ProcessStart
            #ioPM_Inface.ProcessStart := TRUE;

            // Transition to next step: 115
            IF TRUE THEN  // Sequential transition - review XML for actual condition
                #State := STEP_ST10_Flow15_FRobot_3_PickPallet;
            END_IF;

        // ===========================================
        // STEP 115: PickPallet
        // ===========================================
        STEP_ST10_Flow15_FRobot_3_PickPallet:
            // Action Qualifier=R
            // Token: #ioPM_Inface.ProcessComplete
            #ioPM_Inface.ProcessComplete := FALSE;
            // Action Qualifier=S
            // Token: #ioPM_Inface.ProcessStart
            #ioPM_Inface.ProcessStart := TRUE;

            // Transition to next step: 315
            IF TRUE THEN  // Sequential transition - review XML for actual condition
                #State := STEP_ST10_Flow15_FRobot_3_WaitPos3ScanFinish;
            END_IF;

        // ===========================================
        // STEP 315: WaitPos3ScanFinish
        // ===========================================
        STEP_ST10_Flow15_FRobot_3_WaitPos3ScanFinish:
            // No actions in XML

            // Transition to next step: 357
            IF TRUE THEN  // Sequential transition - review XML for actual condition
                #State := STEP_ST10_Flow15_FRobot_3_WaitRobotReachScanPos;
            END_IF;

        // ===========================================
        // STEP 357: WaitRobotReachScanPos
        // ===========================================
        STEP_ST10_Flow15_FRobot_3_WaitRobotReachScanPos:
            // No actions in XML

            // Transition to next step: 361
            IF TRUE THEN  // Sequential transition - review XML for actual condition
                #State := STEP_ST10_Flow15_FRobot_3_StartRobotPressRingPut;
            END_IF;

        // ===========================================
        // STEP 361: StartRobotPressRingPut
        // ===========================================
        STEP_ST10_Flow15_FRobot_3_StartRobotPressRingPut:
            // Action Qualifier=N
            // Token: "KukaRobot3_CtrlDB".sPLCtoROB.User.Cycle.DI277_PressPutRingReq
            "KukaRobot3_CtrlDB".sPLCtoROB.User.Cycle.DI277_PressPutRingReq;

            // Transition to next step: 704
            IF TRUE THEN  // Sequential transition - review XML for actual condition
                #State := STEP_ST10_Flow15_FRobot_3_ReqRobotToMantenPos_1;
            END_IF;

        // ===========================================
        // STEP 704: ReqRobotToMantenPos_1
        // ===========================================
        STEP_ST10_Flow15_FRobot_3_ReqRobotToMantenPos_1:
            // Action Qualifier=N
            // Token: "KukaRobot3_CtrlDB".sPLCtoROB.User.Cycle.DI297_MaintainRequest
            "KukaRobot3_CtrlDB".sPLCtoROB.User.Cycle.DI297_MaintainRequest;

            // Transition to next step: 130
            IF TRUE THEN  // Sequential transition - review XML for actual condition
                #State := STEP_ST10_Flow15_FRobot_3_PickTable;
            END_IF;

        // ===========================================
        // STEP 130: PickTable
        // ===========================================
        STEP_ST10_Flow15_FRobot_3_PickTable:
            // Action Qualifier=R
            // Token: #ioPM_Inface.ProcessComplete
            #ioPM_Inface.ProcessComplete := FALSE;
            // Action Qualifier=S
            // Token: #ioPM_Inface.ProcessStart
            #ioPM_Inface.ProcessStart := TRUE;

            // Transition to next step: 260
            IF TRUE THEN  // Sequential transition - review XML for actual condition
                #State := STEP_ST10_Flow15_FRobot_3_DataMove_3;
            END_IF;

        // ===========================================
        // STEP 260: DataMove_3
        // ===========================================
        STEP_ST10_Flow15_FRobot_3_DataMove_3:
            // Action Qualifier=N
            // Token: "AutoProcessData".B_Press2.RingCode_2 := "AutoProcessData".F_Robot3Grip2.RingCode_2
            "AutoProcessData".B_Press2.RingCode_2 := "AutoProcessData".F_Robot3Grip2.RingCode_2;
            // Action Qualifier=N
            // Token: "AutoProcessData".B_Press2.PartStatus := 420
            "AutoProcessData".B_Press2.PartStatus := 420;

            // Transition to next step: 300
            IF TRUE THEN  // Sequential transition - review XML for actual condition
                #State := STEP_ST10_Flow15_FRobot_3_PickGlueNGProcess;
            END_IF;

        // ===========================================
        // STEP 300: PickGlueNGProcess
        // ===========================================
        STEP_ST10_Flow15_FRobot_3_PickGlueNGProcess:
            // No actions in XML

            // Transition to next step: 326
            IF TRUE THEN  // Sequential transition - review XML for actual condition
                #State := STEP_ST10_Flow15_FRobot_3_StartRobotPickPalletShaft;
            END_IF;

        // ===========================================
        // STEP 326: StartRobotPickPalletShaft
        // ===========================================
        STEP_ST10_Flow15_FRobot_3_StartRobotPickPalletShaft:
            // Action Qualifier=N
            // Token: "KukaRobot3_CtrlDB".sPLCtoROB.User.Cycle.DI241_PickPalletReq
            "KukaRobot3_CtrlDB".sPLCtoROB.User.Cycle.DI241_PickPalletReq;

            // Transition to next step: 749
            IF TRUE THEN  // Sequential transition - review XML for actual condition
                #State := STEP_ST10_Flow15_FRobot_3_NG1_PutProcessFinish;
            END_IF;

        // ===========================================
        // STEP 749: NG1 PutProcessFinish
        // ===========================================
        STEP_ST10_Flow15_FRobot_3_NG1_PutProcessFinish:
            // Action Qualifier=S
            // Token: #ioPM_Inface.ProcessComplete
            #ioPM_Inface.ProcessComplete := TRUE;
            // Action Qualifier=R
            // Token: #ioPM_Inface.ProcessStart
            #ioPM_Inface.ProcessStart := FALSE;

            // Transition to next step: 155
            IF TRUE THEN  // Sequential transition - review XML for actual condition
                #State := STEP_ST10_Flow15_FRobot_3_OKPut;
            END_IF;

        // ===========================================
        // STEP 155: OKPut
        // ===========================================
        STEP_ST10_Flow15_FRobot_3_OKPut:
            // Action Qualifier=R
            // Token: #ioPM_Inface.ProcessComplete
            #ioPM_Inface.ProcessComplete := FALSE;
            // Action Qualifier=S
            // Token: #ioPM_Inface.ProcessStart
            #ioPM_Inface.ProcessStart := TRUE;

            // Transition to next step: 299
            IF TRUE THEN  // Sequential transition - review XML for actual condition
                #State := STEP_ST10_Flow15_FRobot_3_PickPalletFinish;
            END_IF;

        // ===========================================
        // STEP 299: PickPalletFinish
        // ===========================================
        STEP_ST10_Flow15_FRobot_3_PickPalletFinish:
            // Action Qualifier=S
            // Token: #ioPM_Inface.ProcessComplete
            #ioPM_Inface.ProcessComplete := TRUE;
            // Action Qualifier=R
            // Token: #ioPM_Inface.ProcessStart
            #ioPM_Inface.ProcessStart := FALSE;

            // Transition to next step: 350
            IF TRUE THEN  // Sequential transition - review XML for actual condition
                #State := STEP_ST10_Flow15_FRobot_3_MagnScanNGProcess;
            END_IF;

